	bSeqAbort					:BOOL;		(*Function Abort By Manager*)
	bSeqHomingRequest			:BOOL;		(*FUNCTION Homing Requested BY Manager OR Internal Functions*)
	bSeqWaitOnRequest			:BOOL;		(*Function In Valide State Avaiting For Request Command*)
	bSeqRequest					:BOOL;		(*Request Commnad To Start Function Cycle*)

	bSeqIsHoming					: BOOL;
	bSeqInProgress				:BOOL;		(*Function In Progress With Cycle*)
	bSeqComplete				:BOOL;		(*Function Complete Cycle - Flag Set After Every Cycle Finsh*)
	bSeqDone					:BOOL;		(*Function Sequence Finished With Success - Flag Set For One PLC Cycle*)
	bSeqError						: BOOL;
	nSeqErrorID					: UDINT;

	bAutoHomingAllowed			: BOOL;
	bStationHomed					:BOOL;		(*FUNCTION Homed*)
	bStationNotMoving				:BOOL;		(*Function Parts Are Not Moving*)
	bStationInPause				: BOOL;

	bMachineInError				: BOOL;
	bPassthroughMode				:BOOL;

	stBundleTracking				: ST_BundleTrackingRegister_C715;
	bTrackigDataSync				: BOOL;
	bDisableBottomLimit			: BOOL;

	bSynchroMoveActive			: BOOL;

END_STRUCT
END_TYPE

// ---- DUTs/METS/_StationOperational/C715 Tempalate Example/ST_BundleTrackingRegister_C715.TcDUT
TYPE ST_BundleTrackingRegister_C715 :
STRUCT
	bOuterPresent				: BOOL;
	sOuterTimeStamp			: STRING(30);
	bOuterAligned				: BOOL;
	bLabelApplied				: BOOL;		(* TRUE = label has been printed and applied to Outer *)
	bLabelFormed				: BOOL;
	sLabelBarcode				: T_OUTER_Barcode;
	sConfirmationCode 			: T_MaxString;
	bOCVCreated				: BOOL;
	bOACCreated				: BOOL;
	bOuterIsValid				: BOOL;
	bDumpDataReq			: BOOL;
END_STRUCT
END_TYPE

// ---- DUTs/METS/_StationOperational/E_00_StationStateTemplate.TcDUT
TYPE E_00_StationStateTemplate :
(
	SEQ_00_INIT									:=0,
	SEQ_00_ENABLEDEVICES							:=1,
	SEQ_00_HOMING								:=10,
	SEQ_00_MOVETOHOMEPOS_TRY					:=20,
	SEQ_00_MOVETOHOMEPOS_DONE					:=30,
	SEQ_00_HOMED								:=90,
	SEQ_00_READY									:=100,

	SEQ_00_REQACCEPTED							:=110,

(***************************************************************************)
(**)
(***************************************************************************)

	SEQ_00_COMPLETE_TRY							:=340,
	SEQ_00_COMPLETE								:=350


);
END_TYPE

// ---- DUTs/METS/_StationOperational/Manual Machine/E_OuterPrintStationState.TcDUT
TYPE E_OuterPrintStationState :
(
	STATION_SEQ_INIT:=100,
	STATION_SEQ_TRY_HOMING:=110,
	STATION_SEQ_HOMED:=120,
	STATION_SEQ_READY:=130,

	STATION_SEQ_GATE_DOWN_TRY:=140,
	STATION_SEQ_GATE_DOWN_DONE:=150,

	STATION_SEQ_APPLY_LABEL_TRY:=160,
	STATION_SEQ_APPLY_LABEL_DONE:=170,

	STATION_SEQ_GATE_UP_TRY:=180,
	STATION_SEQ_GATE_UP_DONE:=190,

	STATION_SEQ_COMPLETE_TRY:=200,
	STATION_SEQ_COMPLETE:=210


);
END_TYPE

// ---- DUTs/METS/_StationOperational/Manual Machine/ST_OuterPrintStationStruct.TcDUT
TYPE ST_OuterPrintStationStruct :
STRUCT

	eOuterPrintStationState				: 	E_OuterPrintStationState;

	bStationRequest			: 	BOOL;		(*Request Commnad To Start Function Cycle*)
	bStationWaitOnRequest	:	BOOL;		(*Function In Valide State Avaiting For Request Command*)
	bStationInProgress		: 	BOOL;		(*Function In Progress With Cycle*)
	bStationComplete			: 	BOOL;		(*Function Complete Cycle - Flag Set After Every Cycle Finsh*)

	bStationHomingRequest		:	BOOL;		(*FUNCTION Homing Requested BY Manager OR Internal Functions*)
	bStationHomed					: 	BOOL;		(*FUNCTION Homed*)
	bStationDone					:	BOOL;		(*Function Sequence Finished With Success - Flag Set For One PLC Cycle*)
	bStationAbort					: 	BOOL;		(*Function Abort By Manager*)
	bStationInhibit					: BOOL;

	bStationNotMoving			: 	BOOL;		(*Function Parts Are Not Moving*)

	bPassthroughMode						: BOOL;


	eGateCommand		: E_CYLINDER_Position := E_CYLINDER_Position.STOP;

	bGateInPosition					: BOOL;
	bGateRetractedPosition				: BOOL;
	bGateExtendedPosition				: BOOL;
	bGateIsRetracting					: BOOL;
	bGateIsExtending					: BOOL;
	bGatePositionError					: BOOL;

	bOuterAtApplyPosition					: BOOL;
	bApplyLabel							: BOOL;
	bApplyDone							: BOOL;

	bSkipGate							: BOOL;
END_STRUCT
END_TYPE

// ---- DUTs/METS/_StationOperational/SeqCtrl/ST_STATION_Requests.TcDUT
TYPE ST_STATION_Requests :
STRUCT

	bSeqAbort						:BOOL;		(*Function Abort By Manager*)
	bSeqInhibit						: BOOL;		(*in girafe is like bMachineInError*)
	bSeqHomingRequest			:BOOL;		(*FUNCTION Homing Requested BY Manager OR Internal Functions*)
	bSeqWaitOnRequest			:BOOL;		(*Function In Valide State Avaiting For Request Command*)
	bSeqRequest					:BOOL;		(*Request Commnad To Start Function Cycle*)

END_STRUCT
END_TYPE

// ---- DUTs/METS/_StationOperational/SeqCtrl/ST_STATION_Status.TcDUT
TYPE ST_STATION_Status :
STRUCT

	bSeqIsHoming					: BOOL;
	bStationHomed					:BOOL;		(*FUNCTION Homed*)
	bSeqInProgress				:BOOL;		(*Function In Progress With Cycle*)
	bSeqComplete				:BOOL;		(*Function Complete Cycle - Flag Set After Every Cycle Finsh*)
	bSeqDone					:BOOL;		(*Function Sequence Finished With Success - Flag Set For One PLC Cycle*)
	bStationNotMoving				:BOOL;		(*Function Parts Are Not Moving*)

	bSeqError						: BOOL;
	nSeqErrorID					: UDINT;

END_STRUCT
END_TYPE

// ---- DUTs/METS/_StationOperational/ST_00_StationStructTemplate.TcDUT
TYPE ST_00_StationStructTemplate :
STRUCT

	e00SeqState		: E_00_StationStateTemplate;

	REQ				: ST_STATION_Requests;
	STAT				: ST_STATION_Status;

(*Variable examles only*)
(*
	bPassthroughMode			:BOOL;

	stBundleTracking				: ST_BundleTrackingRegister;
	bTrigCamera					: BOOL;
	bCameraDone					: BOOL;


*)

END_STRUCT
END_TYPE

// ---- DUTs/Test_DUTs/ST_DuplicateInfo.TcDUT
TYPE ST_DuplicateInfo :
STRUCT
	value 			: T_MaxString;
	nOuterIndex 	: UINT;
	PackIndex 		: UINT;
END_STRUCT
END_TYPE

// ---- DUTs/Test_DUTs/ST_FBinside.TcDUT
TYPE ST_FBinside :
STRUCT
	aTONs		: ARRAY[1..10] OF TON;
	aTOFs		: ARRAY[1..10] OF TOF;
END_STRUCT
END_TYPE

// ---- DUTs/Test_DUTs/ST_LAB_CaseData.TcDUT
TYPE ST_LAB_CaseData :
STRUCT
	aOuters		: ARRAY[1..50] OF ST_LAB_OuterData;
END_STRUCT
END_TYPE

// ---- DUTs/Test_DUTs/ST_LAB_OuterData.TcDUT
TYPE ST_LAB_OuterData :
STRUCT
	sOuterCode			: T_MaxString;
	nOutersStatus		: INT;
	nOuterRejectID		: UINT;
	
	aPacks				: ARRAY[1..10] OF ST_LAB_PackData;
END_STRUCT
END_TYPE

// ---- DUTs/Test_DUTs/ST_LAB_PackData.TcDUT
TYPE ST_LAB_PackData :
STRUCT
	sPackCode			: T_MaxString;
	nPackStatus			: INT;
	nPackRejectID		: UINT;
END_STRUCT
END_TYPE

// ---- GVLs/CodeAI.TcGVL
{attribute 'Tc2GvlVarNames'}
VAR_GLOBAL
	eCodeAIType							: E_CodeAIType;
	


END_VAR

// ---- GVLs/gConstants.TcGVL
{attribute 'Tc2GvlVarNames'}
//{warning 'CONVERSION MESSAGE: This text contained unprintable characters, that have been deleted'.}
VAR_GLOBAL CONSTANT

	(* sub-folders for  directory *)
	cSYSTEM_FOLDER_LIMIT				: INT :=20;

	(*cBASE_FOLDER_ARR					: ARRAY[1..cSYSTEM_FOLDER_LIMIT] OF T_FolderName :=[
			(*01*)'Bridge\',	(*02*)'Bridge\Archive\',	(*03*)'Bridge\Restore\',
			(*04*)'CAC\',		(*05*)'CAC\Archive\',		(*06*)'CAC\Error\',	(*07*)'CAC\Restore\', 	(*08*)'CAC\Restore\Archive\',
			(*09*)'CHM\',		(*10*)'CHM\Archive\',		(*11*)'CHM\Error\',	(*12*)'CHM\OK\',		(*13*)'CHM\Commissioning_Mode\',
			(*14*)'HMI\',
			(*15*)'KPI\',		(*16*)'KPI\Archive\',		(*17*)'KPI\Shift\',	(*18*)'KPI\ProdOrder\',
			(*19*)'OAC\',		(*20*)'OAC\Error\',
			(*21*)'OCV\',		(*22*)'OCV\Error\',
			(*23*)'OHM\',		(*24*)'OHM\Archive\',		(*25*)'OHM\Error\',	(*26*)'OHM\OK\',		(*27*)'OHM\Pending\',
			(*28*)'PCM\',		(*29*)'PCM\Archive\',		(*30*)'PCM\Error\',	(*31*)'PCM\Incoming\',
			(*32*)'PAC\',
			(*33*)'PHM\',		(*34*)'PHM\Archive\',		(*35*)'PHM\Error\',	(*36*)'PHM\OK\',
			(*37*)'Settings\',	(*38*)'Settings\Backups\',
			(*39*)'Templates\',
			(*40*)'Orca\',
			(*41*)'SystemLog\',
			(*42*)'Cameras\',
			(*43*)'ArchiveDB\'];*)
			
cMETS_CORE_FOLDERS					: ARRAY[1..cSYSTEM_FOLDER_LIMIT] OF T_FolderName :=[
			(*01*)'CHM\',		(*02*)'CHM\Archive\',		(*03*)'CHM\Error\',		(*04*)'CHM\OK\',		(*05*)'CHM\Commissioning_Mode\',	(*06*)'CHM\Restore\',
			(*07*)'PCM\',		(*08*)'PCM\Archive\',		(*09*)'PCM\Error\',		(*10*)'PCM\Incoming\',
			(*11*)'Settings\',	(*12*)'Settings\Backups\',	(*13*)'Settings\Recipe\',
			(*14*)'Cameras\',
			(*15*)'Printers\',	(*16*)'Printers\Templates'];
			
cMETS_AUX_FOLDERS					: ARRAY[1..cSYSTEM_FOLDER_LIMIT] OF T_FolderName :=[
			(*01*)'CAC\',		(*02*)'CAC\Archive\',		(*03*)'CAC\Error\',		(*04*)'CAC\Restored\',
			(*05*)'OAC\',		(*06*)'OAC\Error\',			(*07*)'OAC\Empty\',
			(*08*)'OCV\',		(*09*)'OCV\Error\',			(*10*)'OCV\Empty\',
			(*11*)'SystemLog\',
			(*12*)'ArchiveDB\',
			(*13*)'BridgeApp\Bridge_Core\',
			(*14*)'LoggerApp\Service\',
			(*15*)'WebHMI\',
			(*16*)'DeleteArchiveTool\'];
			
			
	cME_ARCHIVE_ACTION 					: ARRAY[1..3] OF STRING :=[
			(*01*)'Archive', 	(*02*)'DeleteTime', 		(*03*)'DeleteItem'] ;

	cMAX_HMI_DISPLAYS					: INT:=2;
	cMAX_HMI_SERIALCODE_LENGHT			: INT := 33;

	cDISABLE_LOG						: BOOL := FALSE;
	cDISABLE_ALARMS						: BOOL := FALSE;
	cMAX_ALARM_GROUP					: T_PositiveINT:=7;
	cMAX_MESSAGE_NUMBER					: T_PositiveINT:=255;
	cMAX_DISPLAY_ALARMS					: T_PositiveINT := 100;

	cMAX_PACK_INFEED_QUEUE				: T_PositiveINT := 80;  (*IMPORTANT index needs to by grater than max value form aPackCodeMapping20*)
	cMAX_HMI_PACK_INFEED_QUEUE			: T_PositiveINT :=100;	(*must be FIXED 100 for HMI and bigger then cMAX_PACK_INFEED_QUEUE*)

	cMAX_INTERMEDIATE_CODE_QUEUE		: T_PositiveINT := 10;
	(*cMAX_TRACE_UNIT_QUEUE				: UINT := 5;
	cMAX_PACK_REJECTED_QUEUE			: UINT := 30;*)

	cMAX_PACKCODE_LENGHT				: T_PositiveINT := 60;
	cMAX_HMI_PACKCODE_LENGHT			: T_PositiveINT := 67;

	cMAX_PACKS_PER_OUTER				: T_PositiveINT :=10;
	cMAX_HMI_PACKS_PER_OUTER			: T_PositiveINT :=20;	(*must be FIXED 20 for HMI and bigger then cMAX_PACKS_PER_OUTER*)

	cMAX_OUTER_STATUS_QUEUE				: T_PositiveINT := 50;
	cMAX_INFEED_QUEUE					: T_PositiveINT :=100;

	cMAX_OUTERS_PER_CASE 				: T_PositiveINT := 70;
	cMAX_HMI_OUTERS_PER_CASE 			: T_PositiveINT := 100;	(*must be FIXED  100 for HM and bigger then cMAX_OUTERS_PER_CASE*)

	cMAX_PACK_PER_CASE 					: T_PositiveINT := 840;	(*must be cMAX_PACKS_PER_OUTER* cMAX_OUTERS_PER_CASE*)

	cMAX_SIDEFLEX_QUEUE					: T_PositiveINT :=10;
	cMAX_CASE_QUEUE						: T_PositiveINT :=4;
	cMAX_FAILED_CASE_QUEUE				: T_PositiveINT :=10;
	cMAX_VERIFIED_CASE_QUEUE			: T_PositiveINT :=10;
	cMAX_LAST_CASE_BARCODES				: T_PositiveINT := 10;

	cMAX_CHM_PACKID_LENGHT				: T_PositiveINT := 60;
	cMAX_CHM_OUTERID_LENGHT				: T_PositiveINT := 60;
	cMAX_CHM_CASEID_LENGHT				: T_PositiveINT := 25;

	cSHIFTNUMBER						: T_PositiveINT := 4;

	cCODE_OVERWIRTTEN					: STRING(12) := '************';
	cCASE_PACKER_REJECT					: STRING := 'CASE_REJECT_BY_CASEPACKER';
	cMAX_REJECT_REASON					: T_PositiveINT := 80;
	cXML_HEADER							: STRING :=   '<?xml version="1.0" encoding="utf-8"?>$R$N';

	cPARAMETER_STORAGE_SIZE				: T_PositiveINT := 25;	(*  *)


	cMAX_ETHERCAT_SLAVES				: T_PositiveINT := 63; 	(* tabel start with 0 and 64 elemnts *)
	cMAX_PNOZ_ELEMENTS					: T_PositiveINT := 20;
	cMAX_PROFINET_MASTERS	      		: T_PositiveINT := 2; 		(* Must always be set min to 2*)
	cMAX_PROFINET_DRIVES        		: T_PositiveINT := 8;		(* Must always be set min to 8*)
	cMAX_ANALOG_DRIVERS					: T_PositiveINT := 2; 		(* Must always be set min to 2*)
	cMAX_MC2_DRIVES						: T_PositiveINT := 2;
	cMAX_CYLINDERS						: T_PositiveINT := 12;		(*Must always be set min to 3*)
	cMAX_PRINTER_NUMBER           		: T_PositiveINT := 6;		(*Must always be set min to 6*)
	cMAX_HAND_SCANNERS					: T_PositiveINT := 2; 		(*Must always be set min to 2*)
	cMAX_CAMS							: T_PositiveINT := 1;
	cMAX_ENCODER						: T_PositiveINT := 1;
	cMAX_CAMERA_PROG_NUMBER				: T_PositiveINT := 5;
	cMAX_CAMERA_NUMBER					: T_PositiveINT :=12;		(*Must always be set min to 12*)
	cOUT_CAMERA_GROUP					: T_PositiveINT:=9;
	cCS_CAMERA_GROUP					: T_PositiveINT:=12;
	cPLAS_CAMERA_OFF_DELAY				: TIME:= T#10S;

	cDOT_CHAR 							: T_Char := '.';
	cTAB_CHAR 							: T_Char := '$09';
	cLF_CHAR 							: T_Char := '$0A';
	cCR_CHAR							: T_Char := '$0D';

	cHALF_SECOND						: TIME := t#0.5s;
	cONE_SECOND							: TIME := T#1s;
	cTWO_SECONDS						: TIME := T#2s;
	cTHREE_SECONDS						: TIME := T#3s;
	cFIVE_SECONDS						: TIME := t#5s;
	cTEN_SECONDS						: TIME := t#10s;

	cONE_MINUTE							: TIME := t#1m;
	cFIVE_MINUTES						: TIME := T#5m;
	cONE_HOUR							: TIME := T#1h;

	(* File handling *)
	cFAILED_INVALID_INDEX_GROUP			: DWORD :=  16#702;
	cFAILED_INVALID_INDEX_OFFSET		: DWORD :=  16#703;
	cFAILED_OBJECT_NOT_FOUND			: DWORD :=  16#70C;
	cFAILED_OBJECT_ALREADY_EXIST		: DWORD :=  16#70F;
	cFAILED_NO_MORE_FILE_HANDLES		: DWORD :=  16#716;
	cFAILED_ACCESS_DENIED				: DWORD :=  16#723;
	
	(* File handling *)
	//cFAILED_INVALID_DATA				: DWORD :=  16#703;
	//cFAILED_FILE_NOT_FOUND			: DWORD :=  16#70C;
	//cFAILED_NO_MORE_FILE_HANDLES		: DWORD :=  16#716;
	cMAX_FILE_BUFFER					: T_PositiveINT := 32767;(*10000;*)

	cNUMBER_DEFINED_AI_TYPES			: T_PositiveINT :=14;
	cMAX_VALIDATION_ITEMS				: T_PositiveINT :=10;

	(*cUSE_INTERMEDIATE_BARCODE_VALIDATION	: BOOL := TRUE;*)

	cMAX_CAMERA_TYPES					: T_PositiveINT :=15;

	cACQUISITION_TIMER					: ARRAY[0..cMAX_CAMERA_TYPES] OF TIME :=[
			(*Number of array elemnts must match to number of elemnts in E_SCANNER_DeviceType*)
			(*E_MV_None*)T#0ms,
			(*E_MV_420_FULL*)T#26ms,			(*E_MV_420_HALF*)T#12ms,
			(*E_MV_440SR_FULL*)T#18ms, 		(*E_MV_440SR_HALF*)T#12ms,
			(*E_MV_440HR_FULL*)T#52ms, 		(*E_MV_440HR_HALF*)T#30ms,
			(*E_MV_440UR_FULL*)T#50ms, 		(*E_MV_440UR_HALF*)T#33ms,
			(*E_MV_540S_FULL*)T#24ms, 			(*E_MV_540S_HALF*)T#12ms,
			(*E_MV_540H_FULL*)T#24ms, 			(*E_MV_540H_HALF*)T#12ms,
			(*E_MV_560U_FULL*)T#24ms, 			(*E_MV_560U_HALF*)T#12ms,
			(*E_V_430F_FULL*)T#18ms];


END_VAR

// ---- GVLs/GVL.TcGVL
{attribute 'qualified_only'}
VAR_GLOBAL
	bTriggerButton		AT %I* : BOOL;			
	bTriggerOutput		AT %Q* : BOOL;		


	// Hikrobot Control Commands

	aHikrobotCtrlCommands				: ARRAY[1..20] OF STRING(40) :=[
		(*start user params 0*) 		'<Set,UserStart,0>',
		(*start user params 1*) 		'<Set,UserStart,1>',
		(*start user params 2*) 		'<Set,UserStart,2>',
		(*execute self adjustement*) 	'<Exec,Tune>',
		(*start reading codes*) 		'<Set,Acq,1><Set,UserStart,3>',
		(*stop reading codes*) 			'<Set,Acq,0>',
		(*camera reboot*) 				'<Exec,Reboot>',
		(*camera reboot*) 				'<Get,RunMode>',
		(*camera reboot*) 				'<Set,RunMode,2>',
		(*camera reboot*) 				'<Set,RunMode,0>'
];


	aTCPxStrings						: ARRAY[0..20] OF T_MaxString;
	aTCPxStringsReply					: ARRAY[0..20] OF T_MaxString;

END_VAR

// ---- GVLs/GVL_HIKROBOT_COMMANDS.TcGVL
{attribute 'qualified_only'}
VAR_GLOBAL
END_VAR

// ---- GVLs/GVL_test.TcGVL
{attribute 'qualified_only'}
VAR_GLOBAL
	
	//aCase	: ARRAY[1..3] OF ST_LAB_OuterData ;
	stCase		:	ST_LAB_CaseData; 
	stCaseFull	:	ST_LAB_CaseData; 

	
	nMax_Outers			: UINT := 50;
	nMax_Packs			: UINT := 10;


	
// 	aInputArray		: ARRAY[1..3, 1..3] OF T_MaxString := [ 
// 	['PACK01OUTER1', 'PACK02OUTER1', 'PACK03OUTER1'],
// 	['PACK01OUTER2', 'PACK02OUTER2', 'PACK03OUTER2'],
// 	['PACK01OUTER3', 'PACK02OUTER3', 'PACK03OUTER3']
// 	];


	stFBinside		: ST_FBinside;

END_VAR

// ---- POUs/PRG_TEST.TcPOU
PROGRAM PRG_TEST
VAR
	//fbCaseDuplicatCheckTests			: FB_CASE_DuplicatCheckTests;
	//fbCaseDuplicateUpdateToDBTests	: FB_CASE_DuplicateUpdateToDBTests;
	//fbCaseFinaliseDataTests				: FB_CASE_FinaliseDataTests;
	//fbCaseInitialiseData_Test 			: FB_CASE_InitialiseDataTests;
	fbCaseValidateContentTests		: FB_CASE_ValidateContentTests;
	
END_VAR

//===================================================
//UNIT TEST EXECUTION

TcUnit.RUN();

//===================================================
//MANUAL TEST EXECUTION

PRG_CASE_DuplicatCheckManual();
PRG_CASE_DuplicateUpdateToDBManual();
PRG_CASE_FinaliseDataManual();
PRG_CASE_InitialiseDataManual();
PRG_CASE_ValidateContentManual();



//===================================================
//TESTS for FB references
//PRG_Reference_POU();

END_PROGRAM

// ---- POUs/TcUnit/FB_CASE_ValidateContentTests/FB_CASE_ValidateContentTests.TcPOU
FUNCTION_BLOCK FB_CASE_ValidateContentTests EXTENDS TcUnit.FB_TestSuite

VAR
	
(* General data *)
	stCTDateTime_tests					: ST_SYSTEM_DateTime;	
	stProductInstruction_tests			: ST_PCM_Status;
	nSecquentionalCounter_tests			: UDINT;
	stCodeInfo_Outer_tests				: ST_CodeInfo;
	stCaseRejectReasons_tests			: ST_RejectReasonsForCase;
	stRejectReasonsForOuter_tests		: ST_RejectReasonsForOuter;
	stOuterDataNotFound_tests			: ST_RejectItems;

(* 01.Main tests container *)

	stProductInstruction_test_0101		: ST_PCM_Status;
	stCACData_test_0101 				: ST_CAC_Data;
		
	stCACData_tests 					: ST_CAC_Data;
(* 02.DataConsistancy tests container *)
	stProductInstruction_test_0201		: ST_PCM_Status;
	stCACData_test_0201 				: ST_CAC_Data;
	sRejectCode_test_0201				: T_MaxString;
	
	stProductInstruction_test_0202		: ST_PCM_Status;
	stCACData_test_0202 				: ST_CAC_Data;
	sRejectCode_test_0202				: T_MaxString;	
	
	
	stProductInstruction_test_0203		: ST_PCM_Status;
	stCACData_test_0203 				: ST_CAC_Data;
	sRejectCode_test_0203				: T_MaxString;
	
	stProductInstruction_test_0204		: ST_PCM_Status;
	stCACData_test_0204 				: ST_CAC_Data;
	sRejectCode_test_0204				: T_MaxString;

	
	stProductInstruction_test_0205		: ST_PCM_Status;
	stCACData_test_0205 				: ST_CAC_Data;
	sRejectCode_test_0205				: T_MaxString;
	
	stProductInstruction_test_0206		: ST_PCM_Status;
	stCACData_test_0206 				: ST_CAC_Data;
	sRejectCode_test_0206				: T_MaxString;

(* 03.NumberOfOuters tests container *)
	stProductInstruction_test_0301		: ST_PCM_Status;
	stCACData_test_0301 				: ST_CAC_Data;
	sRejectCode_test_0301				: T_MaxString;
	
	stProductInstruction_test_0302		: ST_PCM_Status;
	stCACData_test_0302 				: ST_CAC_Data;
	sRejectCode_test_0302				: T_MaxString;
	
	stProductInstruction_test_0303		: ST_PCM_Status;
	stCACData_test_0303 				: ST_CAC_Data;
	sRejectCode_test_0303				: T_MaxString;
	
(* 04.OuterAggrDissable tests container *)
	stProductInstruction_test_0401		: ST_PCM_Status;
	stCACData_test_0401 				: ST_CAC_Data;
	sRejectCode_test_0401				: T_MaxString;
	
	stProductInstruction_test_0402		: ST_PCM_Status;
	stCACData_test_0402 				: ST_CAC_Data;
	sRejectCode_test_0402				: T_MaxString;

(* 05.OuterAggrEnable tests container *)
	stProductInstruction_test_0501		: ST_PCM_Status;
	stCACData_test_0501 				: ST_CAC_Data;
	sRejectCode_test_0501				: T_MaxString;
	
	stProductInstruction_test_0502		: ST_PCM_Status;
	stCACData_test_0502 				: ST_CAC_Data;
	sRejectCode_test_0502				: T_MaxString;

(* 06.DuplicateHandler tests container *)
	
	stProductInstruction_test_0601		: ST_PCM_Status;
	stCACData_test_0601 				: ST_CAC_Data;
	sRejectCode_test_0601				: T_MaxString;
	
	stCACData_test_0602 				: ST_CAC_Data;
	stProductInstruction_test_0602		: ST_PCM_Status;
	sRejectCode_test_0602				: T_MaxString;
	
(* 07.OACmissing tests container *)
	
	stProductInstruction_test_0701		: ST_PCM_Status;
	stCACData_test_0701 				: ST_CAC_Data;
	sRejectCode_test_0701				: T_MaxString;
	
	stCACData_test_0702 				: ST_CAC_Data;
	stProductInstruction_test_0702		: ST_PCM_Status;
	sRejectCode_test_0702				: T_MaxString;
	
	sRejectCode_tets					: T_MaxString;
	
END_VAR


//==============================================================
//01.Main
//==============================================================
main01_bExecuteFalseNoAction();
//==============================================================
//02.DataConsistancy
//==============================================================
dataConsistancy01_NumOfOutersWrong();
dataConsistancy02_NumOfOutersExceedcMAX_Outers();
dataConsistancy03_ValidationCodeNotFoundInInfeedQueue();
dataConsistancy04_OuterCodeVal_IndexErrorFound();
dataConsistancy05_NumberOfOutersToSmall();
dataConsistancy06_NumberOfOutersToBig();

//==============================================================
//03.NumberOfOuters
//==============================================================
numberOfOuters01_ValueToLittlebErrorTrue();
numberOfOuters02_ValueGraterErrorTrue();
numberOfOuters03_ValueToLittlebErrorTrueRejectCodeWright();

//==============================================================
//04.OuterAggrDissable
//==============================================================
outerAggrDissable01_sRejectCodeOK();

//==============================================================
//05.OuterAggrEnable
//==============================================================
outerAggrEnable01_PacksPerOuterZero();
outerAggrEnable02_PacksPerCaseZero();


//==============================================================
//06.DuplicatesHandler
//==============================================================
duplicateHandler01_OuterDuplicatebErrorTrue();
duplicateHandler02_PackDuplicatebErrorTrue();

//==============================================================
//07.OACmissing
//==============================================================
oacMissing01nErrorID21();

METHOD INTERNAL dataConsistancy01_NumOfOutersWrong
VAR
	//fbCaseTest			: FB_CASE_ValidateContent;
	bDone				: BOOL;
	bBusy				: BOOL;
	bError				: BOOL;
	nErrorID 			: UDINT;
	nValidationIndex	: INT;
	
	eLastState			: E_CAC_State;
			
END_VAR

VAR_INST
	fbCaseTest0201				: FB_CASE_ValidateContent;
	rTrig0201					: R_TRIG;
	nCycles0201					: INT;
	
END_VAR

//Data initialization
TestInit(stCACData:= stCACData_test_0201, stProductInstruction:= stProductInstruction_test_0201);

//Change some data for test scenario below
stCACData_test_0201.NumberOfOuters := stCACData_test_0201.NumberOfOuters - 2;
	
TcUnit.TEST('dataConsistancy01_NumOfOutersWrong');


fbCaseTest0201(
	bExecute:= TRUE, 
	bIsDuplicateOuters:= FALSE, 
	bIsDuplicatePacks:= FALSE, 
	stCTDateTime:= stCTDateTime_tests, 
	stOuterDataNotFound:= stRejectReasonsForOuter_tests.stOuterDataNotFound, 
	stProductInstruction:= stProductInstruction_test_0201, 
	nSecquentionalCounter:= nSecquentionalCounter_tests, 
	stCodeInfo_Outer:= stCodeInfo_Outer_tests, 
	stCaseRejectReasons:= stCaseRejectReasons_tests, 
	stCACData:= stCACData_test_0201, 
	bDone=> bDone, 
	bBusy=> bBusy, 
	bError=> bError, 
	nErrorID=> nErrorID, 
	sRejectCode=> sRejectCode_test_0201, 
	nValidationIndex=> nValidationIndex
);
	
rTrig0201(CLK:= fbCaseTest0201.bDone);
nCycles0201 := nCycles0201 + 1;	

IF rTrig0201.Q THEN	
		
	AssertEquals_BOOL(Expected 	:= TRUE,
					  Actual 	:= bError,
					  Message 	:= 'Wrong number of outers not detected'
	);
	
	AssertEquals_STRING(Expected := 'XXVAL048XX',
						Actual := TO_STRING(fbCaseTest0201.sRejectCode),
						Message := 'Wrong value of nErrorID'
	);
	
	TEST_FINISHED();
	
ELSIF nCycles0201 > 50 THEN
	
	AssertTrue(Condition := TRUE,
			   Message 	 := 'Timeout dataConsistancy01_NumOfOutersWrong'
	);	 
	TEST_FINISHED();
END_IF
END_METHOD

METHOD INTERNAL dataConsistancy02_NumOfOutersExceedcMAX_Outers
VAR
	//fbCaseTest			: FB_CASE_ValidateContent;
	bDone				: BOOL;
	bBusy				: BOOL;
	bError				: BOOL;
	nErrorID 			: UDINT;
	nValidationIndex	: INT;
	
	eLastState			: E_CAC_State;
			
END_VAR

VAR_INST
	fbCaseTest0202				: FB_CASE_ValidateContent;
	rTrig0202					: R_TRIG;
	nCycles0202					: INT;
	
END_VAR

//Data initialization
TestInit(stCACData:= stCACData_test_0202, stProductInstruction:= stProductInstruction_test_0202);

//Change some data for test scenario below
stCACData_test_0202.NumberOfOuters := - 1;
	
TcUnit.TEST('dataConsistancy02_NumOfOutersExceedcMAX_Outers');


fbCaseTest0202(
	bExecute:= TRUE, 
	bIsDuplicateOuters:= FALSE, 
	bIsDuplicatePacks:= FALSE, 
	stCTDateTime:= stCTDateTime_tests, 
	stOuterDataNotFound:= stRejectReasonsForOuter_tests.stOuterDataNotFound, 
	stProductInstruction:= stProductInstruction_test_0202, 
	nSecquentionalCounter:= nSecquentionalCounter_tests, 
	stCodeInfo_Outer:= stCodeInfo_Outer_tests, 
	stCaseRejectReasons:= stCaseRejectReasons_tests, 
	stCACData:= stCACData_test_0202, 
	bDone=> bDone, 
	bBusy=> bBusy, 
	bError=> bError, 
	nErrorID=> nErrorID, 
	sRejectCode=> sRejectCode_test_0202, 
	nValidationIndex=> nValidationIndex
);
	
rTrig0202(CLK:= fbCaseTest0202.bDone);
nCycles0202 := nCycles0202 + 1;	

IF rTrig0202.Q THEN	
		
	AssertEquals_UDINT(Expected := 11,
                   	   Actual 	:= fbCaseTest0202.nErrorID,
                   	   Message 	:= 'nErrorID value wrong');
	
	TEST_FINISHED();
	
ELSIF nCycles0202 > 50 THEN
	
	AssertTrue(Condition := TRUE,
			   Message 	 := 'Timeout dataConsistancy02_NumOfOutersExceedcMAX_Outers'
	);	 
	TEST_FINISHED();
END_IF
END_METHOD

METHOD INTERNAL dataConsistancy03_ValidationCodeNotFoundInInfeedQueue
VAR
	//fbCaseTest			: FB_CASE_ValidateContent;
	bDone				: BOOL;
	bBusy				: BOOL;
	bError				: BOOL;
	nErrorID 			: UDINT;
	nValidationIndex	: INT;
	
	eLastState			: E_CAC_State;
			
END_VAR

VAR_INST
	fbCaseTest0203				: FB_CASE_ValidateContent;
	rTrig0203					: R_TRIG;
	nCycles0203					: INT;
	
END_VAR

//Data initialization
TestInit(stCACData:= stCACData_test_0203, stProductInstruction:= stProductInstruction_test_0203);

//Change some data for test scenario below
stCACData_test_0203.NumberOfOuters := - 2;
	
TcUnit.TEST('dataConsistancy03_ValidationCodeNotFoundInInfeedQueue');


fbCaseTest0203(
	bExecute:= TRUE, 
	bIsDuplicateOuters:= FALSE, 
	bIsDuplicatePacks:= FALSE, 
	stCTDateTime:= stCTDateTime_tests, 
	stOuterDataNotFound:= stRejectReasonsForOuter_tests.stOuterDataNotFound, 
	stProductInstruction:= stProductInstruction_test_0203, 
	nSecquentionalCounter:= nSecquentionalCounter_tests, 
	stCodeInfo_Outer:= stCodeInfo_Outer_tests, 
	stCaseRejectReasons:= stCaseRejectReasons_tests, 
	stCACData:= stCACData_test_0203, 
	bDone=> bDone, 
	bBusy=> bBusy, 
	bError=> bError, 
	nErrorID=> nErrorID, 
	sRejectCode=> sRejectCode_test_0203, 
	nValidationIndex=> nValidationIndex
);
	
rTrig0203(CLK:= fbCaseTest0203.bDone);
nCycles0203 := nCycles0203 + 1;	

IF rTrig0203.Q THEN	
		
	AssertEquals_UDINT(Expected := 12,
                   	   Actual 	:= fbCaseTest0203.nErrorID,
                   	   Message 	:= 'nErrorID value wrong');
	
	TEST_FINISHED();
	
ELSIF nCycles0203 > 50 THEN
	
	AssertTrue(Condition := TRUE,
			   Message 	 := 'Timeout dataConsistancy03_ValidationCodeNotFoundInInfeedQueue'
	);	 
	TEST_FINISHED();
END_IF
END_METHOD

METHOD INTERNAL dataConsistancy04_OuterCodeVal_IndexErrorFound
VAR
	//fbCaseTest			: FB_CASE_ValidateContent;
	bDone				: BOOL;
	bBusy				: BOOL;
	bError				: BOOL;
	nErrorID 			: UDINT;
	nValidationIndex	: INT;
	
	eLastState			: E_CAC_State;
			
END_VAR

VAR_INST
	fbCaseTest0204				: FB_CASE_ValidateContent;
	rTrig0204					: R_TRIG;
	nCycles0204					: INT;
	
END_VAR

//Data initialization
TestInit(stCACData:= stCACData_test_0204, stProductInstruction:= stProductInstruction_test_0204);

//Change some data for test scenario below
stCACData_test_0204.NumberOfOuters := - 3;
	
TcUnit.TEST('dataConsistancy04_OuterCodeVal_IndexErrorFound');


fbCaseTest0204(
	bExecute:= TRUE, 
	bIsDuplicateOuters:= FALSE, 
	bIsDuplicatePacks:= FALSE, 
	stCTDateTime:= stCTDateTime_tests, 
	stOuterDataNotFound:= stRejectReasonsForOuter_tests.stOuterDataNotFound, 
	stProductInstruction:= stProductInstruction_test_0204, 
	nSecquentionalCounter:= nSecquentionalCounter_tests, 
	stCodeInfo_Outer:= stCodeInfo_Outer_tests, 
	stCaseRejectReasons:= stCaseRejectReasons_tests, 
	stCACData:= stCACData_test_0204, 
	bDone=> bDone, 
	bBusy=> bBusy, 
	bError=> bError, 
	nErrorID=> nErrorID, 
	sRejectCode=> sRejectCode_test_0204, 
	nValidationIndex=> nValidationIndex
);
	
rTrig0204(CLK:= fbCaseTest0204.bDone);
nCycles0204 := nCycles0204 + 1;	

IF rTrig0204.Q THEN	
		
	AssertEquals_UDINT(Expected := 13,
                   	   Actual 	:= fbCaseTest0204.nErrorID,
                   	   Message 	:= 'nErrorID value wrong');
	
	TEST_FINISHED();
	
ELSIF nCycles0204 > 50 THEN
	
	AssertTrue(Condition := TRUE,
			   Message 	 := 'Timeout dataConsistancy04_OuterCodeVal_IndexErrorFound'
	);	 
	TEST_FINISHED();
END_IF
END_METHOD

METHOD INTERNAL dataConsistancy05_NumberOfOutersToSmall
VAR
	//fbCaseTest			: FB_CASE_ValidateContent;
	bDone				: BOOL;
	bBusy				: BOOL;
	bError				: BOOL;
	nErrorID 			: UDINT;
	nValidationIndex	: INT;
	
	eLastState			: E_CAC_State;
			
END_VAR

VAR_INST
	fbCaseTest0205				: FB_CASE_ValidateContent;
	rTrig0205					: R_TRIG;
	nCycles0205					: INT;
	
END_VAR

//Data initialization
TestInit(stCACData:= stCACData_test_0205, stProductInstruction:= stProductInstruction_test_0205);

//Change some data for test scenario below
stCACData_test_0205.NumberOfOuters := 25;
	
TcUnit.TEST('dataConsistancy05_NumberOfOutersToSmall');


fbCaseTest0205(
	bExecute:= TRUE, 
	bIsDuplicateOuters:= FALSE, 
	bIsDuplicatePacks:= FALSE, 
	stCTDateTime:= stCTDateTime_tests, 
	stOuterDataNotFound:= stRejectReasonsForOuter_tests.stOuterDataNotFound, 
	stProductInstruction:= stProductInstruction_test_0205, 
	nSecquentionalCounter:= nSecquentionalCounter_tests, 
	stCodeInfo_Outer:= stCodeInfo_Outer_tests, 
	stCaseRejectReasons:= stCaseRejectReasons_tests, 
	stCACData:= stCACData_test_0205, 
	bDone=> bDone, 
	bBusy=> bBusy, 
	bError=> bError, 
	nErrorID=> nErrorID, 
	sRejectCode=> sRejectCode_test_0205, 
	nValidationIndex=> nValidationIndex
);
	
rTrig0205(CLK:= fbCaseTest0205.bDone);
nCycles0205 := nCycles0205 + 1;	

IF rTrig0205.Q THEN	
		
	AssertEquals_UDINT(Expected := 14,
                   	   Actual 	:= fbCaseTest0205.nErrorID,
                   	   Message 	:= 'nErrorID value wrong');
	
	TEST_FINISHED();
	
ELSIF nCycles0205 > 50 THEN
	
	AssertTrue(Condition := TRUE,
			   Message 	 := 'Timeout dataConsistancy05_NumberOfOutersToSmall'
	);	 
	TEST_FINISHED();
END_IF
END_METHOD

METHOD INTERNAL dataConsistancy06_NumberOfOutersToBig
VAR
	//fbCaseTest			: FB_CASE_ValidateContent;
	bDone				: BOOL;
	bBusy				: BOOL;
	bError				: BOOL;
	nErrorID 			: UDINT;
	nValidationIndex	: INT;
	
	eLastState			: E_CAC_State;
			
END_VAR

VAR_INST
	fbCaseTest0206				: FB_CASE_ValidateContent;
	rTrig0206					: R_TRIG;
	nCycles0206					: INT;
	
END_VAR

//Data initialization
TestInit(stCACData:= stCACData_test_0206, stProductInstruction:= stProductInstruction_test_0206);

//Change some data for test scenario below
stCACData_test_0206.NumberOfOuters := 69;
	
TcUnit.TEST('dataConsistancy06_NumberOfOutersToBig');


fbCaseTest0206(
	bExecute:= TRUE, 
	bIsDuplicateOuters:= FALSE, 
	bIsDuplicatePacks:= FALSE, 
	stCTDateTime:= stCTDateTime_tests, 
	stOuterDataNotFound:= stRejectReasonsForOuter_tests.stOuterDataNotFound, 
	stProductInstruction:= stProductInstruction_test_0206, 
	nSecquentionalCounter:= nSecquentionalCounter_tests, 
	stCodeInfo_Outer:= stCodeInfo_Outer_tests, 
	stCaseRejectReasons:= stCaseRejectReasons_tests, 
	stCACData:= stCACData_test_0206, 
	bDone=> bDone, 
	bBusy=> bBusy, 
	bError=> bError, 
	nErrorID=> nErrorID, 
	sRejectCode=> sRejectCode_test_0206, 
	nValidationIndex=> nValidationIndex
);
	
rTrig0206(CLK:= fbCaseTest0206.bDone);
nCycles0206 := nCycles0206 + 1;	

IF rTrig0206.Q THEN	
		
	AssertEquals_UDINT(Expected := 15,
                   	   Actual 	:= fbCaseTest0206.nErrorID,
                   	   Message 	:= 'nErrorID value wrong');
	
	TEST_FINISHED();
	
ELSIF nCycles0206 > 50 THEN
	
	AssertTrue(Condition := TRUE,
			   Message 	 := 'Timeout dataConsistancy06_NumberOfOutersToBig'
	);	 
	TEST_FINISHED();
END_IF
END_METHOD

METHOD INTERNAL duplicateHandler01_OuterDuplicatebErrorTrue
VAR
	//fbCaseTest			: FB_CASE_ValidateContent;
	bDone				: BOOL;
	bBusy				: BOOL;
	bError				: BOOL;
	nErrorID 			: UDINT;
	nValidationIndex	: INT;
	
	eLastState			: E_CAC_State;
			
END_VAR

VAR_INST
	fbCaseTest0601				: FB_CASE_ValidateContent;
	fTrig						: F_TRIG;	
	rTrig						: R_TRIG;
	nCycles						: INT;
	
END_VAR

//Data initialization
TestInit(stCACData:= stCACData_test_0601, stProductInstruction:= stProductInstruction_test_0601);

//Change some data for test scenario below
//stCACData_test_0303.NumberOfOuters := 51;

	
TcUnit.TEST('duplicateHandler01_OuterDuplicatebErrorTrue');



fbCaseTest0601(
	bExecute:= TRUE, 
	bIsDuplicateOuters:= TRUE, 
	bIsDuplicatePacks:= FALSE, 
	stCTDateTime:= stCTDateTime_tests, 
	stOuterDataNotFound:= stRejectReasonsForOuter_tests.stOuterDataNotFound, 
	stProductInstruction:= stProductInstruction_test_0601, 
	nSecquentionalCounter:= nSecquentionalCounter_tests, 
	stCodeInfo_Outer:= stCodeInfo_Outer_tests, 
	stCaseRejectReasons:= stCaseRejectReasons_tests, 
	stCACData:= stCACData_test_0601, 
	bDone=> bDone, 
	bBusy=> bBusy, 
	bError=> bError, 
	nErrorID=> nErrorID, 
	sRejectCode=> sRejectCode_tets, 
	nValidationIndex=> nValidationIndex
);
	
rTrig(CLK:= fbCaseTest0601.bDone);
nCycles := nCycles + 1;	

IF rTrig.Q THEN	
		
	AssertEquals_BOOL(Expected 	:= TRUE,
					  Actual 	:= bError,
					  Message 	:= 'Outer duplicate did not call error'
	);
	
	AssertEquals_UDINT(Expected := 1,
                   	   Actual 	:= fbCaseTest0601.nErrorID,
                   	   Message 	:= 'Wrong nErrorID on outer duplicate'
	);
	
	TEST_FINISHED();
	
ELSIF nCycles > 50 THEN
	
	AssertTrue(Condition := TRUE,
			   Message 	 := 'Timeout duplicateHandler01_OuterDuplicatebErrorTrue'
	);	 
	TEST_FINISHED();
END_IF
END_METHOD

METHOD INTERNAL duplicateHandler02_PackDuplicatebErrorTrue
VAR
	//fbCaseTest			: FB_CASE_ValidateContent;
	bDone				: BOOL;
	bBusy				: BOOL;
	bError				: BOOL;
	nErrorID 			: UDINT;
	nValidationIndex	: INT;
	
	eLastState			: E_CAC_State;
			
END_VAR

VAR_INST
	fbCaseTest0602				: FB_CASE_ValidateContent;
	fTrig						: F_TRIG;	
	rTrig						: R_TRIG;
	nCycles						: INT;
	
END_VAR

//Data initialization
TestInit(stCACData:= stCACData_test_0602, stProductInstruction:= stProductInstruction_test_0602);

//Change some data for test scenario below

	
TcUnit.TEST('duplicateHandler02_PackDuplicatebErrorTrue');


fbCaseTest0602(
	bExecute:= TRUE, 
	bIsDuplicateOuters:= FALSE, 
	bIsDuplicatePacks:= TRUE, 
	stCTDateTime:= stCTDateTime_tests, 
	stOuterDataNotFound:= stRejectReasonsForOuter_tests.stOuterDataNotFound, 
	stProductInstruction:= stProductInstruction_test_0602, 
	nSecquentionalCounter:= nSecquentionalCounter_tests, 
	stCodeInfo_Outer:= stCodeInfo_Outer_tests, 
	stCaseRejectReasons:= stCaseRejectReasons_tests, 
	stCACData:= stCACData_test_0602, 
	bDone=> bDone, 
	bBusy=> bBusy, 
	bError=> bError, 
	nErrorID=> nErrorID, 
	sRejectCode=> sRejectCode_tets, 
	nValidationIndex=> nValidationIndex
);
	
rTrig(CLK:= fbCaseTest0602.bDone);
nCycles := nCycles + 1;	

IF rTrig.Q THEN	
		
	AssertEquals_BOOL(Expected 	:= TRUE,
					  Actual 	:= bError,
					  Message 	:= 'Pack duplicate did not call error'
	);
	
	AssertEquals_UDINT(Expected := 1,
                   	   Actual 	:= fbCaseTest0602.nErrorID,
                   	   Message 	:= 'Wrong nErrorID on pack duplicate'
	);
	
	TEST_FINISHED();
	
ELSIF nCycles > 50 THEN
	
	AssertTrue(Condition := TRUE,
			   Message 	 := 'Timeout duplicateHandler02_PackDuplicatebErrorTrue'
	);	 
	TEST_FINISHED();
END_IF
END_METHOD

METHOD INTERNAL main01_bExecuteFalseNoAction
VAR
	//fbCaseTest			: FB_CASE_ValidateContent;
	bDone				: BOOL;
	bBusy				: BOOL;
	bError				: BOOL;
	nErrorID 			: UDINT;
	nValidationIndex	: INT;
	
	eLastState			: E_CAC_State;
			
END_VAR

VAR_INST
	fbCaseTest0101				: FB_CASE_ValidateContent;
	fTrig						: F_TRIG;	
	rTrig						: R_TRIG;
	nCycles						: INT;
	
END_VAR

//Data initialization
TestInit(stCACData:= stCACData_test_0101, stProductInstruction:= stProductInstruction_test_0101);

//Change some data for test scenario below

	
TcUnit.TEST('main01_bExecuteFalseNoAction');


fbCaseTest0101(
	bExecute:= FALSE, 
	bIsDuplicateOuters:= FALSE, 
	bIsDuplicatePacks:= FALSE, 
	stCTDateTime:= stCTDateTime_tests, 
	stOuterDataNotFound:= stRejectReasonsForOuter_tests.stOuterDataNotFound, 
	stProductInstruction:= stProductInstruction_test_0101, 
	nSecquentionalCounter:= nSecquentionalCounter_tests, 
	stCodeInfo_Outer:= stCodeInfo_Outer_tests, 
	stCaseRejectReasons:= stCaseRejectReasons_tests, 
	stCACData:= stCACData_test_0101, 
	bDone=> bDone, 
	bBusy=> bBusy, 
	bError=> bError, 
	nErrorID=> nErrorID, 
	sRejectCode=> sRejectCode_tets, 
	nValidationIndex=> nValidationIndex
);
	
rTrig(CLK:= fbCaseTest0101.bDone);
nCycles := nCycles + 1;	

		
AssertEquals_BOOL(Expected 	:= FALSE,
				  Actual 	:= fbCaseTest0101.bError,
				  Message 	:= 'FB no executed wrong output'
);

AssertEquals_BOOL(Expected 	:= FALSE,
				  Actual 	:= fbCaseTest0101.bDone,
				  Message 	:= 'B no executed wrong output'
);

TEST_FINISHED();
END_METHOD

METHOD INTERNAL numberOfOuters01_ValueToLittlebErrorTrue
VAR
	//fbCaseTest			: FB_CASE_ValidateContent;
	bDone				: BOOL;
	bBusy				: BOOL;
	bError				: BOOL;
	nErrorID 			: UDINT;
	nValidationIndex	: INT;
	
	eLastState			: E_CAC_State;
			
END_VAR

VAR_INST
	fbCaseTest0301				: FB_CASE_ValidateContent;
	fTrig0301						: F_TRIG;
	nCycles0301						: INT;
	
END_VAR

//Data initialization
TestInit(stCACData:= stCACData_test_0301, stProductInstruction:= stProductInstruction_test_0301);

//Change some data for test scenario below
stCACData_test_0301.NumberOfOuters := 45;
	


TcUnit.TEST('numberOfOuters01_ValueToLittlebErrorTrue');

fbCaseTest0301(
	bExecute:= TRUE, 
	bIsDuplicateOuters:= FALSE, 
	bIsDuplicatePacks:= FALSE, 
	stCTDateTime:= stCTDateTime_tests, 
	stOuterDataNotFound:= stRejectReasonsForOuter_tests.stOuterDataNotFound, 
	stProductInstruction:= stProductInstruction_test_0301, 
	nSecquentionalCounter:= nSecquentionalCounter_tests, 
	stCodeInfo_Outer:= stCodeInfo_Outer_tests, 
	stCaseRejectReasons:= stCaseRejectReasons_tests, 
	stCACData:= stCACData_test_0301, 
	bDone=> bDone, 
	bBusy=> bBusy, 
	bError=> bError, 
	nErrorID=> nErrorID, 
	sRejectCode=> sRejectCode_test_0301, 
	nValidationIndex=> nValidationIndex
);

fTrig0301(CLK:= fbCaseTest0301.bBusy);
nCycles0301 := nCycles0301 + 1;	

IF fTrig0301.Q AND nCycles0301 <= 50 THEN	
	
	AssertEquals_BOOL(Expected := TRUE,
					  Actual := fbCaseTest0301.bError,
					  Message := 'Numbers of outer wrong value didnt call error'
	);
	
	AssertEquals_STRING(Expected := 'XXVAL045XX',
						Actual := TO_STRING(fbCaseTest0301.sRejectCode),
						Message := 'Wrong value of nErrorID'
	);
	
	AssertEquals_INT(Expected := 45,
					 Actual := stCACData_test_0301.NumberOfOuters,
					 Message := 'INT Values differ'
	);	
	
	TEST_FINISHED();
	
ELSIF nCycles0301 > 50 THEN
	
	AssertTrue(Condition := TRUE,
			   Message := 'Timeout CASE loop within FB_CASE_Validation'
	);	 

	
	TEST_FINISHED();
END_IF
END_METHOD

METHOD INTERNAL numberOfOuters02_ValueGraterErrorTrue
VAR
	
	bDone				: BOOL;
	bBusy				: BOOL;
	bError				: BOOL;
	nErrorID 			: UDINT;
	nValidationIndex	: INT;
	
	eLastState			: E_CAC_State;
	
		
END_VAR

VAR_INST
	
	fbCaseTest0302				: FB_CASE_ValidateContent;
	fTrig0302						: F_TRIG;
	nCycles0302						: INT;
	
END_VAR

//Data initialization
TestInit(stCACData:= stCACData_test_0302, stProductInstruction:= stProductInstruction_test_0302);

//Change some data for test scenario below
stCACData_test_0302.NumberOfOuters := 79;

	
TcUnit.TEST('numberOfOuters02_ValueGraterErrorTrue');


fbCaseTest0302(
	bExecute:= TRUE, 
	bIsDuplicateOuters:= FALSE, 
	bIsDuplicatePacks:= FALSE, 
	stCTDateTime:= stCTDateTime_tests, 
	stOuterDataNotFound:= stRejectReasonsForOuter_tests.stOuterDataNotFound, 
	stProductInstruction:= stProductInstruction_test_0302, 
	nSecquentionalCounter:= nSecquentionalCounter_tests, 
	stCodeInfo_Outer:= stCodeInfo_Outer_tests, 
	stCaseRejectReasons:= stCaseRejectReasons_tests, 
	stCACData:= stCACData_test_0302, 
	bDone=> bDone, 
	bBusy=> bBusy, 
	bError=> bError, 
	nErrorID=> nErrorID, 
	sRejectCode=> sRejectCode_test_0302, 
	nValidationIndex=> nValidationIndex
);
	
fTrig0302(CLK:= fbCaseTest0302.bBusy);
nCycles0302 := nCycles0302 + 1;	

IF fTrig0302.Q AND nCycles0302 <= 50 THEN	
		
	AssertEquals_BOOL(Expected := TRUE,
					  Actual := fbCaseTest0302.bError,
					  Message := 'Numbers of outer wrong value didnt call error'
	);
	
	AssertEquals_STRING(Expected := 'XXVAL079XX',
						Actual := TO_STRING(fbCaseTest0302.sRejectCode),
						Message := 'Wrong value of sRejectCode'
	);
	
	TEST_FINISHED();
	
ELSIF nCycles0302 > 50 THEN
	
	AssertTrue(Condition := TRUE,
			   Message 	 := 'Timeout numberOfOuters02_ValueGraterErrorTrue'
	);	 
	
	TEST_FINISHED();
END_IF
END_METHOD

METHOD INTERNAL numberOfOuters03_ValueToLittlebErrorTrueRejectCodeWright
VAR
	//fbCaseTest			: FB_CASE_ValidateContent;
	bDone				: BOOL;
	bBusy				: BOOL;
	bError				: BOOL;
	nErrorID 			: UDINT;
	nValidationIndex	: INT;
	
	eLastState			: E_CAC_State;
			
END_VAR

VAR_INST
	fbCaseTest0303				: FB_CASE_ValidateContent;
	fTrig						: F_TRIG;
	nCycles						: INT;
	
END_VAR

//Data initialization
TestInit(stCACData:= stCACData_test_0303, stProductInstruction:= stProductInstruction_test_0303);

//Change some data for test scenario below
stCACData_test_0303.NumberOfOuters := 51;

	
TcUnit.TEST('numberOfOuters03_ValueToLittlebErrorTrueRejectCodeWright');


fbCaseTest0303(
	bExecute:= TRUE, 
	bIsDuplicateOuters:= FALSE, 
	bIsDuplicatePacks:= FALSE, 
	stCTDateTime:= stCTDateTime_tests, 
	stOuterDataNotFound:= stRejectReasonsForOuter_tests.stOuterDataNotFound, 
	stProductInstruction:= stProductInstruction_test_0301, 
	nSecquentionalCounter:= nSecquentionalCounter_tests, 
	stCodeInfo_Outer:= stCodeInfo_Outer_tests, 
	stCaseRejectReasons:= stCaseRejectReasons_tests, 
	stCACData:= stCACData_test_0303, 
	bDone=> bDone, 
	bBusy=> bBusy, 
	bError=> bError, 
	nErrorID=> nErrorID, 
	sRejectCode=> sRejectCode_test_0303, 
	nValidationIndex=> nValidationIndex
);
	
fTrig(CLK:= fbCaseTest0303.bBusy);
nCycles := nCycles + 1;	

IF fTrig.Q THEN	
		
	AssertEquals_BOOL(Expected := TRUE,
					  Actual := fbCaseTest0303.bError,
					  Message := 'Numbers of outer wrong value didnt call error'
	);
	
	AssertEquals_STRING(Expected := 'XXVAL051XX',
						Actual := TO_STRING(fbCaseTest0303.sRejectCode),
						Message := 'Wrong value of sRejectCode'
	);
	
	TEST_FINISHED();
	
ELSIF nCycles > 50 THEN
	
	AssertTrue(Condition := TRUE,
			   Message 	 := 'Timeout numberOfOuters03_ValueToLittlebErrorTrueRejectCodeWright'
	);	 
	
	TEST_FINISHED();
END_IF
END_METHOD

METHOD INTERNAL oacMissing01nErrorID21
VAR
	//fbCaseTest			: FB_CASE_ValidateContent;
	bDone				: BOOL;
	bBusy				: BOOL;
	bError				: BOOL;
	nErrorID 			: UDINT;
	nValidationIndex	: INT;
	bCompare			: BOOL;
	
	eLastState			: E_CAC_State;
			
END_VAR

VAR_INST
	fbCaseTest0701				: FB_CASE_ValidateContent;
	fTrig0701					: F_TRIG;	
	rTrig0701					: R_TRIG;
	nCycles0701					: INT;
	
END_VAR

//Data initialization
TestInit(stCACData:= stCACData_test_0701, stProductInstruction:= stProductInstruction_test_0701);

//Change some data for test scenario below
stCACData_test_0701.Outer[5].OuterRejectID := 207;
stProductInstruction_test_0701.nCaseAcceptanceLevelOuters := 60;
stProductInstruction_test_0701.nOuterAcceptanceLevelPacks := 100;
stProductInstruction_test_0701.nCaseAcceptanceLevelPacks  := 100;
	
TcUnit.TEST('oacMissing01nErrorID21');


fbCaseTest0701(
	bExecute:= TRUE, 
	bIsDuplicateOuters:= FALSE, 
	bIsDuplicatePacks:= FALSE, 
	stCTDateTime:= stCTDateTime_tests, 
	stOuterDataNotFound:= stRejectReasonsForOuter_tests.stOuterDataNotFound, 
	stProductInstruction:= stProductInstruction_test_0701, 
	nSecquentionalCounter:= nSecquentionalCounter_tests, 
	stCodeInfo_Outer:= stCodeInfo_Outer_tests, 
	stCaseRejectReasons:= stCaseRejectReasons_tests, 
	stCACData:= stCACData_test_0701, 
	bDone=> bDone, 
	bBusy=> bBusy, 
	bError=> bError, 
	nErrorID=> nErrorID, 
	sRejectCode=> sRejectCode_tets, 
	nValidationIndex=> nValidationIndex
);
	
rTrig0701(CLK:= fbCaseTest0701.bDone);
nCycles0701 := nCycles0701 + 1;	



IF rTrig0701.Q THEN	
	
	bCompare := (stCACData_test_0701.CaseRejectID = stCaseRejectReasons_tests.stOACError.nRejectID);
	
	AssertEquals_BOOL(Expected 	:= TRUE,
					  Actual 	:= bError,
					  Message 	:= 'Pack duplicate did not call error'
	);
	
	AssertEquals_UDINT(Expected := 21,
                   	   Actual 	:= fbCaseTest0701.nErrorID,
                   	   Message 	:= 'Wrong nErrorID on OAC missing'
	);
	
	AssertEquals_BOOL(Expected 	:= TRUE,
					  Actual 	:= bCompare,
					  Message 	:= 'CaseRejectID wrong value'
	);	
	
	TEST_FINISHED();
	
ELSIF nCycles0701 > 50 THEN
	
	AssertTrue(Condition := FALSE,
			   Message 	 := 'Timeout oacMissing01nErrorID21'
	);	 
	TEST_FINISHED();
END_IF
END_METHOD

METHOD INTERNAL outerAggrDissable01_sRejectCodeOK
VAR
	//fbCaseTest			: FB_CASE_ValidateContent;
	bDone				: BOOL;
	bBusy				: BOOL;
	bError				: BOOL;
	nErrorID 			: UDINT;
	nValidationIndex	: INT;
	
	eLastState			: E_CAC_State;
			
END_VAR

VAR_INST
	fbCaseTest0401				: FB_CASE_ValidateContent;
	rTrig0401					: R_TRIG;
	nCycles0401					: INT;
	
END_VAR

//Data initialization
TestInit(stCACData:= stCACData_test_0401, stProductInstruction:= stProductInstruction_test_0401);

//Change some data for test scenario below
stCACData_test_0401.CodingAndTrackingMode := 6;
	
TcUnit.TEST('outerAggrDissable01_sRejectCodeOK');


fbCaseTest0401(
	bExecute:= TRUE, 
	bIsDuplicateOuters:= FALSE, 
	bIsDuplicatePacks:= FALSE, 
	stCTDateTime:= stCTDateTime_tests, 
	stOuterDataNotFound:= stOuterDataNotFound_tests, 
	stProductInstruction:= stProductInstruction_test_0401, 
	nSecquentionalCounter:= nSecquentionalCounter_tests, 
	stCodeInfo_Outer:= stCodeInfo_Outer_tests, 
	stCaseRejectReasons:= stCaseRejectReasons_tests, 
	stCACData:= stCACData_test_0401, 
	bDone=> bDone, 
	bBusy=> bBusy, 
	bError=> bError, 
	nErrorID=> nErrorID, 
	sRejectCode=> sRejectCode_test_0401, 
	nValidationIndex=> nValidationIndex
);
	
rTrig0401(CLK:= fbCaseTest0401.bDone);
nCycles0401 := nCycles0401 + 1;	

IF rTrig0401.Q THEN	
	
	AssertEquals_STRING(Expected := 'OK',
						Actual := TO_STRING(fbCaseTest0401.sRejectCode),
						Message := 'Wrong value of nErrorID'
	);
	
	
	TEST_FINISHED();
	
ELSIF nCycles0401 > 50 THEN
	
	AssertTrue(Condition := TRUE,
			   Message 	 := 'Timeout outerAggrDissable01_sRejectCodeOK'
	);	 
	TEST_FINISHED();
END_IF
END_METHOD

METHOD INTERNAL outerAggrEnable01_PacksPerOuterZero
VAR
	//fbCaseTest			: FB_CASE_ValidateContent;
	bDone				: BOOL;
	bBusy				: BOOL;
	bError				: BOOL;
	nErrorID 			: UDINT;
	nValidationIndex	: INT;
	
	eLastState			: E_CAC_State;
			
END_VAR

VAR_INST
	fbCaseTest0501				: FB_CASE_ValidateContent;
	rTrig0501					: R_TRIG;
	nCycles0501					: INT;
	
END_VAR

//Data initialization
TestInit(stCACData:= stCACData_test_0501, stProductInstruction:= stProductInstruction_test_0501);

//Change some data for test scenario below
stCACData_test_0501.CodingAndTrackingMode := 8;
stProductInstruction_test_0501.nPacksPerOuter := 0;
	
TcUnit.TEST('outerAggrEnable01_PacksPerOuterZero');


fbCaseTest0501(
	bExecute:= TRUE, 
	bIsDuplicateOuters:= FALSE, 
	bIsDuplicatePacks:= FALSE, 
	stCTDateTime:= stCTDateTime_tests, 
	stOuterDataNotFound:= stRejectReasonsForOuter_tests.stOuterDataNotFound, 
	stProductInstruction:= stProductInstruction_test_0501, 
	nSecquentionalCounter:= nSecquentionalCounter_tests, 
	stCodeInfo_Outer:= stCodeInfo_Outer_tests, 
	stCaseRejectReasons:= stCaseRejectReasons_tests, 
	stCACData:= stCACData_test_0501, 
	bDone=> bDone, 
	bBusy=> bBusy, 
	bError=> bError, 
	nErrorID=> nErrorID, 
	sRejectCode=> sRejectCode_test_0501, 
	nValidationIndex=> nValidationIndex
);
	
rTrig0501(CLK:= fbCaseTest0501.bDone);
nCycles0501 := nCycles0501 + 1;	

IF rTrig0501.Q THEN	
	
	AssertEquals_BOOL(Expected 	:= TRUE,
					  Actual 	:= bError,
					  Message 	:= 'Wrong number of outers not detected'
	);

	AssertEquals_UDINT(Expected := 10,
                   	   Actual 	:= fbCaseTest0501.nErrorID,
                   	   Message 	:= 'nErrorID value wrong'
	);
	
	
	TEST_FINISHED();
	
ELSIF nCycles0501 > 50 THEN
	
	AssertTrue(Condition := TRUE,
			   Message 	 := 'Timeout outerAggrEnable01_PacksPerOuterZero'
	);	 
	TEST_FINISHED();
END_IF
END_METHOD

METHOD INTERNAL outerAggrEnable02_PacksPerCaseZero
VAR
	//fbCaseTest			: FB_CASE_ValidateContent;
	bDone				: BOOL;
	bBusy				: BOOL;
	bError				: BOOL;
	nErrorID 			: UDINT;
	nValidationIndex	: INT;
	
	eLastState			: E_CAC_State;
			
END_VAR

VAR_INST
	fbCaseTest0502				: FB_CASE_ValidateContent;
	rTrig0502					: R_TRIG;
	nCycles0502					: INT;
	
END_VAR

//Data initialization
TestInit(stCACData:= stCACData_test_0502, stProductInstruction:= stProductInstruction_test_0502);

//Change some data for test scenario below
stCACData_test_0502.CodingAndTrackingMode := 8;
stProductInstruction_test_0502.nPacksPerCase := 0;
	
TcUnit.TEST('outerAggrEnable02_PacksPerCaseZero');


fbCaseTest0502(
	bExecute:= TRUE, 
	bIsDuplicateOuters:= FALSE, 
	bIsDuplicatePacks:= FALSE, 
	stCTDateTime:= stCTDateTime_tests, 
	stOuterDataNotFound:= stRejectReasonsForOuter_tests.stOuterDataNotFound, 
	stProductInstruction:= stProductInstruction_test_0502, 
	nSecquentionalCounter:= nSecquentionalCounter_tests, 
	stCodeInfo_Outer:= stCodeInfo_Outer_tests, 
	stCaseRejectReasons:= stCaseRejectReasons_tests, 
	stCACData:= stCACData_test_0502, 
	bDone=> bDone, 
	bBusy=> bBusy, 
	bError=> bError, 
	nErrorID=> nErrorID, 
	sRejectCode=> sRejectCode_test_0502, 
	nValidationIndex=> nValidationIndex
);
	
rTrig0502(CLK:= fbCaseTest0502.bDone);
nCycles0502 := nCycles0502 + 1;	

IF rTrig0502.Q THEN	
	
	AssertEquals_BOOL(Expected 	:= TRUE,
					  Actual 	:= bError,
					  Message 	:= 'Wrong number of outers not detected'
	);

	AssertEquals_UDINT(Expected := 10,
                   	   Actual 	:= fbCaseTest0502.nErrorID,
                   	   Message 	:= 'nErrorID value wrong'
	);
	
	
	TEST_FINISHED();
	
ELSIF nCycles0502 > 50 THEN
	
	AssertTrue(Condition := TRUE,
			   Message 	 := 'Timeout outerAggrEnable02_PacksPerCaseZero'
	);	 
	TEST_FINISHED();
END_IF
END_METHOD

METHOD PRIVATE TestInit : BOOL
VAR_IN_OUT
	stProductInstruction	: ST_PCM_Status;
	stCACData 				: ST_CAC_Data;
END_VAR

VAR	
	rTrigDataInit		: R_TRIG;
	bDataInit			: BOOL;
	iOuter				: INT;
	iPack				: INT;
	sPackNum			: STRING;
	sOuterNum			: STRING;
	sPackCode			: STRING;
END_VAR

VAR_OUTPUT
	bDone				: BOOL;
END_VAR

//MEMSET(ADR(stCACData), 16#00, SIZEOF(stCACData));	

stProductInstruction.nOutersPerCase 	:= 50;
stProductInstruction.nPacksPerOuter		:= 10;
stProductInstruction.nPacksPerCase		:= 500;
stProductInstruction.nOpMode			:= 11;
stProductInstruction.sRetailSKU			:= '1234567';
stProductInstruction.nAcceptanceLevel 	:= 10;

stCACData.NumberOfOuters			:= stProductInstruction.nOutersPerCase;
stCACData.CodingAndTrackingMode		:= stProductInstruction.nOpMode;
stCACData.RetailSKU					:= stProductInstruction.sRetailSKU;

FOR iOuter := 1 TO stProductInstruction.nOutersPerCase DO
	(* Outer number z zerami *)
	sOuterNum := F_StringAddPrefix(INT_TO_STRING(iOuter),2,'0');

	stCACData.Outer[iOuter].Barcode    				:= CONCAT('OUTER', sOuterNum);
	stCACData.Outer[iOuter].NumberOfPacks 			:= stProductInstruction.nPacksPerOuter;
	stCACData.Outer[iOuter].NumberOfLinkedPacks 	:= stProductInstruction.nPacksPerOuter;
	stCACData.Outer[iOuter].AcceptanceLevel 		:= stProductInstruction.nAcceptanceLevel;
	stCACData.Outer[iOuter].CodingAndTrackingMode	:= stProductInstruction.nOpMode;
	stCACData.Outer[iOuter].OuterRejectCode			:= 'OK';

	FOR iPack := 1 TO stProductInstruction.nPacksPerOuter DO
		(* Pack number dwucyfrowy z zerami *)
		sPackNum := F_StringAddPrefix(INT_TO_STRING(iPack),2,'0');			
		(* Sklej pack code *)
		sPackCode := CONCAT(CONCAT('PACK', sPackNum), CONCAT('OUTER', sOuterNum));
		
		(* Write Pack Barcodes / Data*)
		stCACData.Outer[iOuter].PackCode[iPack]				:= sPackCode;
		stCACData.Outer[iOuter].PackCodeStatus[iPack]		:= 5;
		stCACData.Outer[iOuter].PackRejectID[iPack]			:= 0;			
		stCACData.Outer[iOuter].PackRejectCode[iPack]		:= 'OK';			
		stCACData.Outer[iOuter].PackCodeStatus[iPack].5 	:= TRUE;
		
		
		IF iPack = 1 THEN
			stCACData.Outer[iOuter].AggregationCodes[1]	:= stCACData.Outer[iOuter].PackCode[iPack];
		END_IF
		IF iPack = 2 THEN
			stCACData.Outer[iOuter].AggregationCodes[2]	:= stCACData.Outer[iOuter].PackCode[iPack];
		END_IF
	END_FOR
END_FOR	

stCACData.Outer[3].OuterCodeStatus.5 	:= TRUE;
stCACData.Outer[4].OuterCodeStatus.5	:= TRUE;
END_METHOD

END_FUNCTION_BLOCK

// ---- POUs/FinaliseCaseData/FB_CASE_ValidateContent.TcPOU
FUNCTION_BLOCK FB_CASE_ValidateContent
VAR_INPUT
	bExecute 					: BOOL;
	stCTDateTime				: ST_SYSTEM_DateTime;	(* CaseTrace date/time structure *)
END_VAR
VAR_IN_OUT

	stProductInstruction		: ST_PCM_Status;
	nSecquentionalCounter		: UDINT;
	stCodeInfo_Outer			: ST_CodeInfo;
	stCaseRejectReasons			: ST_RejectReasonsForCase;
	stCACData 					: ST_CAC_Data;
END_VAR
VAR_OUTPUT
	bDone 						: BOOL;
	bBusy						: BOOL;
	bError						: BOOL;
	nErrorID 					: UDINT;

	sRejectCode					: T_MaxString;
	nValidationIndex			: INT;

END_VAR
VAR
	fbExecute						: R_TRIG;
	eState						: E_CAC_STATE;
	eErrorState					: E_CAC_STATE;

	(*nIndex						: INT;*)

	//bValQtyOver				: BOOL;

	(*fbValidateCaseLabel				: FB_CODE_ValidateExplicitCode;*)
	nOutGTIN					: INT;
	nOutBand					: INT;
	nRetailSKU					: INT;
	nSerialCode					: INT;
	nTotalInvalide				: INT;

	fbValidateOuter				: FB_CODE_ValidateExplicitCode;
	nValidOACData				: INT;

	(*fbValidatePack					: FB_CODE_ValidateExplicitCode;*)
	nOuterIndex					: INT;
	nPackIndex					: INT;
	nValidPackData					: INT;
	//nIndex2: T_PositiveINT;
	//nIndex3: T_PositiveINT;

	aStatusErrorVal					: ARRAY[0..10] OF STRING(10);
	aRejectCodePointer     		   	: ARRAY[0..10] OF STRING(10);
END_VAR

(* rising edge of bExecute *)
fbExecute(CLK:= bExecute);

CASE eState OF

	E_CAC_IDLE:

		(* validate stCACData *)
		IF fbExecute.Q THEN

			(* update outputs *)
			bDone := FALSE;
			bBusy := TRUE;
			bError := FALSE;
			nErrorID := 0;

			MEMSET(ADR(aStatusErrorVal), 16#00, SIZEOF(aStatusErrorVal));
			MEMSET(ADR(aRejectCodePointer), 16#00, SIZEOF(aRejectCodePointer));

			(* clear outputs *)
			sRejectCode 		:= '';
			nValidationIndex	:= 0;

			eState := E_CAC_VALIDATECASE;

		(* bExecute has been reset *)
		ELSIF bExecute = FALSE THEN

			(* clear outputs *)
			bDone := FALSE;
			bBusy := FALSE;
			bError := FALSE;

		END_IF

	(* validate Case data *)
	E_CAC_VALIDATECASE:

		(* Outers in Case is correct *)
		IF stCACData.NumberOfOuters = stProductInstruction.nOutersPerCase THEN

			(* Outer aggregation enabled *)
			IF stCACData.CodingAndTrackingMode >= 7 THEN

				eState := E_CAC_VALIDATEOUTER;

			(* OAC data disabled *)
			ELSE
				eState := E_CAC_DONE;
			END_IF

		(* invalid Case *)
		ELSE

			(* update status *)
			bError := TRUE;
			eErrorState := eState;

			(* no validation code read *)
			IF stCACData.NumberOfOuters = -1 THEN

				(* error code *)
				nErrorID := 11;

				(* reset nNumberOfOuters to 0 and generate reject string *)
				stCACData.NumberOfOuters := 0;

				stCACData.CaseRejectCode 	:= stCaseRejectReasons.stCaseNoCaseData.sMetsDisplayCode;
				stCACData.CaseRejectID 		:= stCaseRejectReasons.stCaseNoCaseData.nRejectID;
				
			(* validation code not found in sInfeedQueue *)
			ELSIF stCACData.NumberOfOuters = -2 THEN

				(* error code *)
				nErrorID := 12;

				(* reset nNumberOfOuters to 0 and generate reject string *)
				stCACData.NumberOfOuters := 0;

				aStatusErrorVal[0] 		:= F_StringAddPrefix(INT_TO_STRING(stCACData.NumberOfOuters),2,'0');
				aRejectCodePointer[0] 	:= 'nn';

				stCACData.CaseRejectCode 	:= F_CODE_AssignValToStringWithPrefix(stCaseRejectReasons.stValError.sMetsDisplayCode, aStatusErrorVal, aRejectCodePointer, 3, '0');
				stCACData.CaseRejectID 		:= stCaseRejectReasons.stValError.nRejectID;

				(*eState := E_CAC_DONE;*)

			ELSIF stCACData.NumberOfOuters = -3 THEN

				(* error code *)
				nErrorID := 13;

				(* reset nNumberOfOuters to 0 and generate reject string *)
				stCACData.NumberOfOuters := stProductInstruction.nOutersPerCase;

				aStatusErrorVal[0] 		:= F_StringAddPrefix(INT_TO_STRING(stCACData.NumberOfOuters),2,'0');
				aRejectCodePointer[0] 	:= 'nn';

				stCACData.CaseRejectCode 	:= F_CODE_AssignValToStringWithPrefix(stCaseRejectReasons.stValError.sMetsDisplayCode, aStatusErrorVal, aRejectCodePointer, 3, '0');
				stCACData.CaseRejectID 		:= stCaseRejectReasons.stValError.nRejectID;

				(*eState := E_CAC_DONE;*)

			(* incorrect number of Outers *)
			ELSE

				aStatusErrorVal[0] 		:= F_StringAddPrefix(INT_TO_STRING(stCACData.NumberOfOuters),2,'0');
				aRejectCodePointer[0] 	:= 'nn';

				stCACData.CaseRejectCode 	:= F_CODE_AssignValToStringWithPrefix(stCaseRejectReasons.stValError.sMetsDisplayCode, aStatusErrorVal, aRejectCodePointer, 3, '0');
				stCACData.CaseRejectID 		:= stCaseRejectReasons.stValError.nRejectID;

				(* >=1 Outer(s) missed by Infeed camera *)
				IF stCACData.NumberOfOuters < stProductInstruction.nOutersPerCase THEN

					(* error code *)
					nErrorID := 14;

				(* >=1 Outer(s) physically removed from Infeed queue *)
				ELSE
					(* error code *)
					nErrorID := 15;
				END_IF
			END_IF

			eState := E_CAC_DONE;
		END_IF

	(* validate RetailSKU for each Outer *)
	E_CAC_VALIDATEOUTER:

		(* initialise counters *)
		nOutGTIN		:= 0;
		nOutBand		:= 0;
		nRetailSKU 		:= 0;
		nSerialCode 	:= 0;
		nTotalInvalide	:= 0;

		(* for each Outer *)
		FOR nOuterIndex := 1 TO stCACData.NumberOfOuters DO

			fbValidateOuter(	sFullCode := stCACData.Outer[nOuterIndex].Barcode,
							stCodeInfo := stCodeInfo_Outer,
							stProductInstruction := stProductInstruction);

			IF fbValidateOuter.bGtinOK  THEN

				(* Outer has valid GTIN *)
				nOutGTIN := nOutGTIN + 1;
			END_IF

			IF fbValidateOuter.bBrandOK  THEN

				(* Outer has valid GTIN *)
				nOutBand := nOutBand + 1;
			END_IF

			IF fbValidateOuter.bSerialCodeOK  THEN

				(* Outer has valid SerialCode *)
				nSerialCode := nSerialCode + 1;
			END_IF

			IF fbValidateOuter.bRskuOK  THEN

				(* Outer has valid RetailSKU *)
				nRetailSKU := nRetailSKU + 1;
			END_IF

			IF fbValidateOuter.bValidationOK THEN

				(* Total number of invalide outers - whatever reaso*)
				nTotalInvalide := nTotalInvalide +1;
			END_IF
		END_FOR


		(* all Outers have valid GTIN *)
		IF  nOutGTIN = stProductInstruction.nOutersPerCase THEN
			(* all Outers have valid Brand *)
			IF  nOutBand = stProductInstruction.nOutersPerCase THEN
				(* all Outers have valid RetailSKU *)
				IF  nRetailSKU = stProductInstruction.nOutersPerCase  THEN
					(* all Outers have valid SerialCode *)
					IF  nSerialCode = stProductInstruction.nOutersPerCase THEN
						(*If total invalide Outers inside a case*)
						IF  nTotalInvalide = stProductInstruction.nOutersPerCase THEN
	
							eState := E_CAC_VALIDATEOAC;
	
						ELSE
							(* RejectCode *)
							bError := TRUE;
							nErrorID := 16;
							eErrorState := eState;

							aStatusErrorVal[0] 		:= F_StringAddPrefix(INT_TO_STRING(stCACData.NumberOfOuters - nTotalInvalide),2,'0');
							aRejectCodePointer[0] 	:= 'nn';
						
							stCACData.CaseRejectCode 	:= F_CODE_AssignValToStringWithPrefix(stCaseRejectReasons.stINVError.sMetsDisplayCode, aStatusErrorVal, aRejectCodePointer, 2, '0');
							stCACData.CaseRejectID 		:= stCaseRejectReasons.stINVError.nRejectID;
							
							eState := E_CAC_DONE;

						END_IF
					(* 1 or more Outers have incorrect SerialCode *)
					ELSE
		
						(* RejectCode *)
						bError := TRUE;
						nErrorID := 17;
						eErrorState := eState;
	
						(* generate reject string *)
	
						aStatusErrorVal[0] 		:= F_StringAddPrefix(INT_TO_STRING(stCACData.NumberOfOuters - nSerialCode),2,'0');
						aRejectCodePointer[0] 	:= 'nn';
	
						stCACData.CaseRejectCode 	:= F_CODE_AssignValToStringWithPrefix(stCaseRejectReasons.stOuterSerialError.sMetsDisplayCode, aStatusErrorVal, aRejectCodePointer, 2, '0');
						stCACData.CaseRejectID 		:= stCaseRejectReasons.stOuterSerialError.nRejectID;
					
						eState := E_CAC_DONE;
	
					END_IF
	
				(* 1 or more Outers with invalid RetailSKU *)
				ELSE
		
					(* RejectCode *)
					bError := TRUE;
					nErrorID := 18;
					eErrorState := eState;
		
					(* generate reject string *)
	
					aStatusErrorVal[0] 		:= F_StringAddPrefix(INT_TO_STRING(stCACData.NumberOfOuters - nRetailSKU),2,'0');
					aRejectCodePointer[0] 	:= 'nn';
		
					stCACData.CaseRejectCode 	:= F_CODE_AssignValToStringWithPrefix(stCaseRejectReasons.stOuterRSKUError.sMetsDisplayCode, aStatusErrorVal, aRejectCodePointer, 2, '0');
					stCACData.CaseRejectID 		:= stCaseRejectReasons.stOuterRSKUError.nRejectID;
					
					eState := E_CAC_DONE;
	
				END_IF
			ELSE
				(* RejectCode *)
				bError := TRUE;
				nErrorID := 19;
				eErrorState := eState;
	
				(* generate reject string *)

				aStatusErrorVal[0] 		:= F_StringAddPrefix(INT_TO_STRING(stCACData.NumberOfOuters - nOutBand),2,'0');
				aRejectCodePointer[0] 	:= 'nn';
	
				stCACData.CaseRejectCode 	:= F_CODE_AssignValToStringWithPrefix(stCaseRejectReasons.stOuterBrandError.sMetsDisplayCode, aStatusErrorVal, aRejectCodePointer, 2, '0');
				stCACData.CaseRejectID 		:= stCaseRejectReasons.stOuterBrandError.nRejectID;
				
				eState := E_CAC_DONE;
			END_IF
		ELSE
		(* RejectCode *)
			bError := TRUE;
			nErrorID := 20;
			eErrorState := eState;

			(* generate reject string *)

			aStatusErrorVal[0] 		:= F_StringAddPrefix(INT_TO_STRING(stCACData.NumberOfOuters - nOutGTIN),2,'0');
			aRejectCodePointer[0] 	:= 'nn';

			stCACData.CaseRejectCode 	:= F_CODE_AssignValToStringWithPrefix(stCaseRejectReasons.stOuterGTINError.sMetsDisplayCode, aStatusErrorVal, aRejectCodePointer, 2, '0');
			stCACData.CaseRejectID 		:= stCaseRejectReasons.stOuterGTINError.nRejectID;
			
			eState := E_CAC_DONE;

		END_IF

(* check OAC data was loaded *)
	E_CAC_VALIDATEOAC:

		(* initialise counter *)
		nValidOACData := 0;

		(* for each Outer *)
		FOR nOuterIndex := 1 TO stCACData.NumberOfOuters DO

			IF stCACData.CodingAndTrackingMode = 7 THEN
				(* OAC mode >= CAC mode, OAC data will contain all data required for CAC mode *)
				IF  stCACData.Outer[nOuterIndex].DataSource <>  'NO_R' AND stCACData.Outer[nOuterIndex].CodingAndTrackingMode = stCACData.CodingAndTrackingMode  THEN
					(* count Outers with valid OAC data *)
					nValidOACData := nValidOACData + 1;
				END_IF
			ELSIF stCACData.CodingAndTrackingMode = 11 THEN
			(* CAC mode -> OAC data will contain all data required for CAC mode *)
				IF stCACData.Outer[nOuterIndex].DataSource <>  'NO_R'  AND stCACData.Outer[nOuterIndex].OuterRejectCode = 'OK'  THEN
					(* count Outers with valid OAC data *)
					nValidOACData := nValidOACData + 1;
				END_IF
			END_IF
		END_FOR

		(* all Outers with valid OAC data *)
		IF (nValidOACData *100 ) / stProductInstruction.nOutersPerCase   >=  stProductInstruction.nCaseAcceptanceLevelOuters THEN


			FOR nOuterIndex := 1 TO stCACData.NumberOfOuters DO

				IF stCACData.CodingAndTrackingMode >= 7 THEN
					(* CAC mode -> OAC data will contain all data required for CAC mode *)
						IF stCACData.Outer[nOuterIndex].DataSource =  'NO_R'  THEN

							stCACData.Outer[nOuterIndex].ProductionDate := F_StringWildcard('#YYYYMMDD#', stCTDateTime.sSystemTime);
							stCACData.Outer[nOuterIndex].ProductionTime := F_StringWildcard('#hhmmss#', stCTDateTime.sSystemTime);
							stCACData.Outer[nOuterIndex].ProductionTimeOffset := F_SYSTEM_SystemTimeOffsetToHHMM(stCTDateTime.nSystemTimeOffset);
		
							stCACData.Outer[nOuterIndex].OuterTimeStamp :=F_SYSTEM_SystemTimeAsISO8601(stCTDateTime.sSystemTime, stCTDateTime.sUTCTimeZoneOffset );
							stCACData.Outer[nOuterIndex].RetailSKU := stProductInstruction.sRetailSKU;
							stCACData.Outer[nOuterIndex].OuterMachine.ProductionSite :=  stProductInstruction.sProductionSite;
							stCACData.Outer[nOuterIndex].OuterMachine.ProductionLine := stProductInstruction.sProductionLine;
							stCACData.Outer[nOuterIndex].BatchNumber := stProductInstruction.sBatchNumber;
							stCACData.Outer[nOuterIndex].CodingAndTrackingMode := stProductInstruction.nOpMode;

							stCACData.Outer[nOuterIndex].NumberOfPacks	:=   stProductInstruction.nPacksPerOuter;
							stCACData.Outer[nOuterIndex].AcceptanceLevel	:= 	stProductInstruction.nAcceptanceLevel;

							stCACData.Outer[nOuterIndex].OuterRejectCode := 'OK';
							stCACData.Outer[nOuterIndex].OuterRejectID := 0;
							stCACData.Outer[nOuterIndex].DataSource :=  '3DC';

						ELSIF stCACData.Outer[nOuterIndex].DataSource <>  'NO_R'  AND stCACData.Outer[nOuterIndex].OuterRejectCode <> 'OK' THEN

							stCACData.Outer[nOuterIndex].OuterRejectCode := 'OK';
							stCACData.Outer[nOuterIndex].OuterRejectID := 0;
							stCACData.Outer[nOuterIndex].DataSource :=  '3DCR';
						END_IF
				END_IF
			END_FOR

			eState := E_CAC_VALIDATEPACK;

		(* 1 or more Outers with missing OAC data *)
		ELSE

			(* update status *)
			bError := TRUE;
			nErrorID := 21;
			eErrorState := eState;

			(* generate reject string *)

			aStatusErrorVal[0] 		:= F_StringAddPrefix(INT_TO_STRING(stCACData.NumberOfOuters - nValidOACData),2,'0');
			aRejectCodePointer[0] 	:= 'nn';

			stCACData.CaseRejectCode 	:= F_CODE_AssignValToStringWithPrefix(stCaseRejectReasons.stOACError.sMetsDisplayCode, aStatusErrorVal, aRejectCodePointer, 3, '0');
			stCACData.CaseRejectID 		:= stCaseRejectReasons.stOACError.nRejectID;

			eState := E_CAC_DONE;
		END_IF

	(* check that PackCode data is included with OAC data *)
	E_CAC_VALIDATEPACK:

		(* initialise counter *)
		nValidPackData := 0;

		(* for each Outer *)
		FOR nOuterIndex := 1 TO stCACData.NumberOfOuters DO

			(* count Outers with PackCode data - assume- outer reject station working fine and only good outers in case, NumberOfLinkedPacks= good pack  *)
			nValidPackData := nValidPackData + stCACData.Outer[nOuterIndex].NumberOfLinkedPacks ;

			FOR nPackIndex := 1 TO stCACData.Outer[nOuterIndex].NumberOfPacks DO

				IF stCACData.Outer[nOuterIndex].PackCodeStatus[nPackIndex].1
					AND stCACData.Outer[nOuterIndex].PackCodeStatus[nPackIndex].2
					AND stCACData.Outer[nOuterIndex].PackCodeStatus[nPackIndex].3	THEN

					nValidPackData := -1;
					EXIT;
				END_IF
			END_FOR

			IF nValidPackData = -1 THEN
				EXIT;
			END_IF

		END_FOR

		(* Outers with PackCode data is correct *)
		IF (nValidPackData *100 ) /  stProductInstruction.nPacksPerCase  >=   stProductInstruction.nCaseAcceptanceLevelPacks   THEN

			FOR nOuterIndex := 1 TO stCACData.NumberOfOuters DO

				IF stCACData.Outer[nOuterIndex].NumberOfLinkedPacks = 0 THEN
					stCACData.Outer[nOuterIndex].PackTimeStamp := F_SYSTEM_SystemTimeAsISO8601(stCTDateTime.sSystemTime, stCTDateTime.sUTCTimeZoneOffset );
				END_IF

				FOR nPackIndex := 1 TO stCACData.Outer[nOuterIndex].NumberOfPacks DO
					(*Tolerance do not modify NumberOfLinkedPacks per outer*) (*later, repalce with PackCodeStatus.0*)
					IF  stCACData.Outer[nOuterIndex].PackCode[nPackIndex] = '' THEN

						stCACData.Outer[nOuterIndex].PackCode[nPackIndex] := F_CODE_BATSerializator(stCTDateTime, ePack, TRUE, stProductInstruction, nSecquentionalCounter);
						(* change reject reason to adjust for tolerance *)
						(*additional bit passing to CAC*)
						stCACData.Outer[nOuterIndex].PackCodeStatus[nPackIndex]:=
														F_FiltredSetBitState16(TRUE, 'LOW', 4, TRUE, stCACData.Outer[nOuterIndex].PackCodeStatus[nPackIndex]);

						stCACData.Outer[nOuterIndex].PackRejectCode[nPackIndex] := 'OK';
						stCACData.Outer[nOuterIndex].PackRejectID[nPackIndex]	:= 0;
					END_IF
				END_FOR

				stCACData.Outer[nOuterIndex].NumberOfLinkedPacks := stCACData.Outer[nOuterIndex].NumberOfPacks;

			END_FOR

			eState := E_CAC_DONE;

		ELSIF nValidPackData = -1 THEN

			(* RejectCode *)
			bError := TRUE;
			nErrorID := 23;
			eErrorState := eState;
	
			aStatusErrorVal[0] 		:= 'PK';
			aRejectCodePointer[0] 	:= 'nn';

			stCACData.CaseRejectCode 	:= F_CODE_AssignValToStringWithPrefix(stCaseRejectReasons.stINVError.sMetsDisplayCode, aStatusErrorVal, aRejectCodePointer, 2, '0');
			stCACData.CaseRejectID 		:= stCaseRejectReasons.stINVError.nRejectID;

			eState := E_CAC_DONE;


		(* 1 or more Outers has no PackCode data *)
		ELSE

			(* update status *)
			bError := TRUE;
			nErrorID := 24;
			eErrorState := eState;

			(* generate reject string *)			(* generate reject string *)
			(*stCACData.RejectCode := F_CONCAT3('XXXPACK', F_StringAddPrefix(INT_TO_STRING(stCACData.NumberOfOuters - nValidPackData), 2, '0'), 'XXX');*)

			aStatusErrorVal[0] 		:= F_StringAddPrefix(INT_TO_STRING(stProductInstruction.nPacksPerCase - nValidPackData),2,'0');
			aRejectCodePointer[0] 	:= 'nn';

			stCACData.CaseRejectCode := F_CODE_AssignValToStringWithPrefix(stCaseRejectReasons.stPackNotLinedError.sMetsDisplayCode, aStatusErrorVal, aRejectCodePointer, 3, '0');
			stCACData.CaseRejectID 	 := stCaseRejectReasons.stPackNotLinedError.nRejectID;

			eState := E_CAC_DONE;
		END_IF

	(* complete *)
	E_CAC_DONE:

		(* no error found *)
		IF bError = FALSE THEN

			stCACData.CaseRejectCode 	:= 'OK';
			stCACData.CaseRejectID		:= 0;
		END_IF

		(* update outputs *)
		bBusy := FALSE;
		bDone := TRUE;
		sRejectCode := stCACData.CaseRejectCode;
		nValidationIndex := stCACData.NumberOfOuters;
		
		eState := E_CAC_IDLE;

(* unknown state *)
ELSE

	eState := E_CAC_IDLE;

	(* clear outputs *)
	bDone := FALSE;
	bBusy := FALSE;
	bError := FALSE;

END_CASE

END_FUNCTION_BLOCK

// ---- POUs/_Utilites/METS/Common LIB/08_SOFTWARE LIB/AI Codes And Validation FBs/F_CODE_AssignValToStringWithPrefix.TcPOU
FUNCTION F_CODE_AssignValToStringWithPrefix : T_MaxString
VAR_INPUT
	asRejectReason		: T_MaxString;
	anValue				: ARRAY[0..10] OF STRING(10);
	asPointer          	  		: ARRAY[0..10] OF STRING(10);
	nPrefixSize			: UINT;
	nPrefixValue			: STRING(5);
END_VAR

VAR
	(*bPointerNotFound	           : BOOL;*)
	nCounter				: INT;
	nPointerPos			: INT;
	asAssignedRejectReason	: T_MaxString;
	sValToAssign			: STRING(20);
END_VAR

(* This Function assigns value to predefined Pointer in string.
     Function can assing up to 10 Values
     For ex. string Reject Reason := 'XXDUPn1-n2XX'
     	         nValue := [3, 4], sPointer := ['n1', 'n2']		
	         asRejectReason := 'XXDUP3-4XX'	*)

F_CODE_AssignValToStringWithPrefix := '';

asAssignedRejectReason := asRejectReason;

REPEAT
	nPointerPos := FIND(asAssignedRejectReason, asPointer[nCounter]);
	IF nPointerPos > 0 AND  asPointer[nCounter] <> '' THEN
		sValToAssign :=  F_StringAddPrefix(anValue[nCounter], nPrefixSize, nPrefixValue);
		 asAssignedRejectReason := REPLACE(asAssignedRejectReason, sValToAssign, LEN(asPointer[nCounter]), nPointerPos);
	END_IF;
	nCounter := nCounter + 1;
UNTIL
	nCounter >= 10
END_REPEAT

IF nCounter <> 0 THEN
	F_CODE_AssignValToStringWithPrefix := asAssignedRejectReason;
ELSE
	F_CODE_AssignValToStringWithPrefix := asRejectReason;
END_IF;

END_FUNCTION

// ---- POUs/_Utilites/METS/F_StringWildcard.TcPOU
(* replaces date and time wildcards in string *)
FUNCTION F_StringWildcard : T_MaxString
VAR_INPUT
	strInput		: T_MaxString;	(* string with wildcard markers *)
	sDateTime		: TIMESTRUCT;	(* date/time structure *)
END_VAR
VAR
	fbExtractData	: FB_ExtractString;
	strWildcard		: T_MaxString;
	strData			: STRING(4);
	nCharPos		: INT;
END_VAR
VAR CONSTANT
	arrMonthCode	: ARRAY[0..12] OF STRING(1) :=[ '', 'A', 'B', 'C', 'D', 'E', 'F', 'G', 'H', 'I', 'J', 'K', 'L'];
END_VAR
(*
-------------------------------------------------------------------------------------------------
Date		Version	Author	Comments
-------------------------------------------------------------------------------------------------
13/04/2015	3.00.01	PB		Check for 'MM' and 'M' now checked last, fixes problem where 'M' followed by 'DD' during April will generate corrupt string.
30/01/2015	3.00.00	PB		Initial release.

-------------------------------------------------------------------------------------------------

The following wildcard strings are supported:
YYYY - Year (4 chars)				hh	- hour
YY	 - Year (last 2 chars)			mm	- minute
Y	 - Year (last char only)		ss	- second
MM	 - Month (01-12 = Jan-Dec)		t	- tenth of second
M	 - Month (A-L = Jan-Dec)
DD	 - Date
*)

(* find and extract wildcard string, enclosed by '#' chars *)
fbExtractData(
	bExtractData	:= TRUE,
	nExtractChars	:= 0, 
	strPrefix		:= '#',
	strSuffix		:= '#',
	strString		:= strInput
);

(* wildcard string found *)
IF fbExtractData.bStringFound = TRUE THEN

	(* log wildcard string for modification *)
	strWildcard := fbExtractData.strData;

	(* check for wildcard 'YYYY' *)
	nCharPos := FIND(strWildcard, 'YYYY');
	IF nCharPos > 0 THEN

		(* generate year as 4 chars and replace YYYY *)
		strData := F_StringAddPrefix(WORD_TO_STRING(sDateTime.wYear), 4, '0');
		strWildcard := REPLACE(strWildcard, strData, 4, nCharPos);

	(* wildcard 'YYYY' not found *)
	ELSE

		(* check for wildcard 'YY' *)
		nCharPos := FIND(strWildcard, 'YY');
		IF nCharPos > 0 THEN

			(* generate year as 2 chars and replace YY *)
			strData := F_StringAddPrefix(RIGHT(WORD_TO_STRING(sDateTime.wYear), 2), 2, '0');
			strWildcard := REPLACE(strWildcard, strData, 2, nCharPos);

		(* wildcard 'YY' not found *)
		ELSE
	
			(* check for wildcard 'Y' *)
			nCharPos := FIND(strWildcard, 'Y');
			IF nCharPos > 0 THEN
	
				(* generate year as 1 char and replace Y *)
				strData := RIGHT(WORD_TO_STRING(sDateTime.wYear), 1);
				strWildcard := REPLACE(strWildcard, strData, 1, nCharPos);
			END_IF
		END_IF
	END_IF

	(* check for wildcard 'DD' *)
	nCharPos := FIND(strWildcard, 'DD');
	IF nCharPos > 0 THEN

		(* generate date as 2 chars and replace DD *)
		strData := F_StringAddPrefix(WORD_TO_STRING(sDateTime.wDay), 2, '0');
		strWildcard := REPLACE(strWildcard, strData, 2, nCharPos);
	END_IF

	(* check for wildcard 'hh' *)
	nCharPos := FIND(strWildcard, 'hh');
	IF nCharPos > 0 THEN

		(* generate hour as 2 chars and replace hh *)
		strData := F_StringAddPrefix(WORD_TO_STRING(sDateTime.wHour), 2, '0');
		strWildcard := REPLACE(strWildcard, strData, 2, nCharPos);
	END_IF

	(* check for wildcard 'mm' *)
	nCharPos := FIND(strWildcard, 'mm');
	IF nCharPos > 0 THEN

		(* generate minute as 2 chars and replace mm *)
		strData := F_StringAddPrefix(WORD_TO_STRING(sDateTime.wMinute), 2, '0');
		strWildcard := REPLACE(strWildcard, strData, 2, nCharPos);
	END_IF

	(* check for wildcard 'ss' *)
	nCharPos := FIND(strWildcard, 'ss');
	IF nCharPos > 0 THEN

		(* generate second as 2 chars and replace ss *)
		strData := F_StringAddPrefix(WORD_TO_STRING(sDateTime.wSecond), 2, '0');
		strWildcard := REPLACE(strWildcard, strData, 2, nCharPos);
	END_IF

	(* check for wildcard 't' *)
	nCharPos := FIND(strWildcard, 't');
	IF nCharPos > 0 THEN

		(* generate tenth of second as 1 char and replace t *)
		strData := WORD_TO_STRING(sDateTime.wMilliseconds / 100);
		strWildcard := REPLACE(strWildcard, strData, 1, nCharPos);
	END_IF

	(* check for wildcard 'MM' *)
	nCharPos := FIND(strWildcard, 'MM');
	IF nCharPos > 0 THEN

		(* generate month as 2 chars and replace MM *)
		strData := F_StringAddPrefix(WORD_TO_STRING(sDateTime.wMonth), 2, '0');
		strWildcard := REPLACE(strWildcard, strData, 2, nCharPos);

	(* wildcard 'YYYY' not found *)
	ELSE

		(* check for wildcard 'M' *)
		nCharPos := FIND(strWildcard, 'M');
		IF nCharPos > 0 THEN

			(* generate month as 1 char and replace M *)
			strData := arrMonthCode[sDateTime.wMonth];
			strWildcard := REPLACE(strWildcard, strData, 1, nCharPos);
		END_IF
	END_IF

	(* insert strWildcard back into strInput *)
	F_StringWildcard := INSERT(strInput, strWildcard, TO_INT(fbExtractData.nStartPos) - 1);

(* no wildcard string found *)
ELSE

	(* strInput direct to output without modification *)
	F_StringWildcard := strInput;
END_IF

END_FUNCTION

// ---- POUs/_Utilites/METS/F_SYSTEM_SystemTimeOffsetToHHMM.TcPOU
(* generate time difference between local time and UTC as "+HH:MM" *)
FUNCTION F_SYSTEM_SystemTimeOffsetToHHMM : STRING(6)
VAR_INPUT
	nSystemTimeOffset	: DINT;		(* UTC offset in ms *)
END_VAR
VAR
	nHours				: DINT;
	nMins				: DINT;
END_VAR
(*
-------------------------------------------------------------------------------------------------
Date		Version	Author	Comments
-------------------------------------------------------------------------------------------------
01/08/2014	2.00.00	PB		Initial release

-------------------------------------------------------------------------------------------------
*)

(* convert ms to hours *)
nHours := ABS(nSystemTimeOffset) / 3600000;

(* remove hours and convert remaining ms to mins *)
nMins := (ABS(nSystemTimeOffset) MOD 3600000) / 60000;

(* construct output string as "+HH:MM" or "-HH:MM" *)
F_SYSTEM_SystemTimeOffsetToHHMM := F_CONCAT4(SEL(nSystemTimeOffset < 0, '+', '-'), F_StringAddPrefix(DINT_TO_STRING(nHours), 2, '0'), ':', F_StringAddPrefix(DINT_TO_STRING(nMins), 2, '0'));

END_FUNCTION

// ---- POUs/_Utilites/METS/Concat Function/F_CONCAT4.TcPOU
(* concatenate 4 strings *)
FUNCTION F_CONCAT4 : T_MaxString
VAR_INPUT
	strString1		: T_MaxString;
	strString2		: T_MaxString;
	strString3		: T_MaxString;
	strString4		: T_MaxString;
END_VAR
VAR
END_VAR
(*
-------------------------------------------------------------------------------------------------
Date		Version	Author	Comments
-------------------------------------------------------------------------------------------------
30/01/2015	3.00.00	PB		No change

-------------------------------------------------------------------------------------------------
05/02/2010	1.00.00	PB		Initial release

-------------------------------------------------------------------------------------------------
*)

F_CONCAT4 := CONCAT(strString1, strString2);
F_CONCAT4 := CONCAT(F_CONCAT4, strString3);
F_CONCAT4 := CONCAT(F_CONCAT4, strString4);

END_FUNCTION

// ---- POUs/_Utilites/METS/F_SYSTEM_SystemTimeAsISO8601.TcPOU
(* generate format 2018-08-08T11:46:15.4869506+02:00*)
FUNCTION F_SYSTEM_SystemTimeAsISO8601 : T_ISO8601Time
VAR_INPUT
	sSystemTime			: TIMESTRUCT;
	strUTCTimeZone		: STRING(6);
END_VAR
VAR
	strYear				: STRING(4);
	strMonth				: STRING(2);
	strDay				: STRING(2);
	strMiliseconds			: STRING(3);

	strHour				: STRING(2);
	strMinute				: STRING(2);
	strSecond				: STRING(2);

	strDate				: STRING(10);
	strTime				: STRING(13);

END_VAR

(*Date*)
	strYear:=F_StringAddPrefix(WORD_TO_STRING(sSystemTime.wYear), 4, '0');
	strMonth:=F_StringAddPrefix(WORD_TO_STRING(sSystemTime.wMonth), 2, '0');
	strDay:=F_StringAddPrefix(WORD_TO_STRING(sSystemTime.wDay), 2, '0');

(*Time*)
	strHour:=F_StringAddPrefix(WORD_TO_STRING(sSystemTime.wHour), 2, '0');
	strMinute:=F_StringAddPrefix(WORD_TO_STRING(sSystemTime.wMinute), 2, '0');
	strSecond:=F_StringAddPrefix(WORD_TO_STRING(sSystemTime.wSecond), 2, '0');
	strMiliseconds:=F_StringAddPrefix(WORD_TO_STRING(sSystemTime.wMilliseconds), 3, '0');
(*Print*)


	strDate:=F_CONCAT5(strYear, '-', strMonth, '-', strDay);
	strTime:=F_CONCAT6('T', strHour, ':', strMinute, ':', strSecond);
	strTime:=F_CONCAT3( strTime,'.', strMiliseconds);

	IF strUTCTimeZone = '+00:00' THEN
		F_SYSTEM_SystemTimeAsISO8601:=F_CONCAT3(strDate, strTime, 'Z');
	ELSE
		F_SYSTEM_SystemTimeAsISO8601:=F_CONCAT3(strDate, strTime, strUTCTimeZone);
	END_IF

END_FUNCTION

// ---- POUs/_Utilites/METS/Concat Function/F_CONCAT5.TcPOU
(* concatenate 5 strings *)
FUNCTION F_CONCAT5 : T_MaxString
VAR_INPUT
	strString1		: T_MaxString;
	strString2		: T_MaxString;
	strString3		: T_MaxString;
	strString4		: T_MaxString;
	strString5		: T_MaxString;
END_VAR
VAR
END_VAR
(*
-------------------------------------------------------------------------------------------------
Date		Version	Author	Comments
-------------------------------------------------------------------------------------------------
30/01/2015	3.00.00	PB		No change

-------------------------------------------------------------------------------------------------
05/02/2010	1.00.00	PB		Initial release

-------------------------------------------------------------------------------------------------
*)

F_CONCAT5 := CONCAT(strString1, strString2);
F_CONCAT5 := CONCAT(F_CONCAT5, strString3);
F_CONCAT5 := CONCAT(F_CONCAT5, strString4);
F_CONCAT5 := CONCAT(F_CONCAT5, strString5);

END_FUNCTION

// ---- POUs/_Utilites/METS/Concat Function/F_CONCAT6.TcPOU
(* concatenate 6 strings *)
FUNCTION F_CONCAT6 : T_MaxString
VAR_INPUT
	strString1		: T_MaxString;
	strString2		: T_MaxString;
	strString3		: T_MaxString;
	strString4		: T_MaxString;
	strString5		: T_MaxString;
	strString6		: T_MaxString;
END_VAR
VAR
END_VAR
(*
-------------------------------------------------------------------------------------------------
Date		Version	Author	Comments
-------------------------------------------------------------------------------------------------
30/01/2015	3.00.00	PB		No change

-------------------------------------------------------------------------------------------------
05/02/2010	1.00.00	PB		Initial release

-------------------------------------------------------------------------------------------------
*)

F_CONCAT6 := CONCAT(strString1, strString2);
F_CONCAT6 := CONCAT(F_CONCAT6, strString3);
F_CONCAT6 := CONCAT(F_CONCAT6, strString4);
F_CONCAT6 := CONCAT(F_CONCAT6, strString5);
F_CONCAT6 := CONCAT(F_CONCAT6, strString6);

END_FUNCTION

// ---- POUs/_Utilites/METS/Concat Function/F_CONCAT3.TcPOU
(* concatenate 3 strings *)
FUNCTION F_CONCAT3 : T_MaxString
VAR_INPUT
	strString1		: T_MaxString;
	strString2		: T_MaxString;
	strString3		: T_MaxString;
END_VAR
VAR
END_VAR
(*
-------------------------------------------------------------------------------------------------
Date		Version	Author	Comments
-------------------------------------------------------------------------------------------------
30/01/2015	3.00.00	PB		No change

-------------------------------------------------------------------------------------------------
05/02/2010	1.00.00	PB		Initial release

-------------------------------------------------------------------------------------------------
*)

F_CONCAT3 := CONCAT(strString1, strString2);
F_CONCAT3 := CONCAT(F_CONCAT3, strString3);

END_FUNCTION

// ---- POUs/_Utilites/METS/F_FiltredSetBitState16.TcPOU
(* updates state of specified bit in nWord value *)
FUNCTION F_FiltredSetBitState16 : WORD
VAR_INPUT
	bEnable		: BOOL;		(* set TRUE to update state of target bit in nValue *)
	sFiltrType		: STRING(5);
	nTargetBit		: INT;		(* bit number of bit to be updated (0-15) *)
	nSetState		: BOOL;		(* state to which nTargetBit should be set *)
	nValue			: WORD;	(* value in which target bit should be updated *)
END_VAR
VAR
	nMaskValue	: WORD;
END_VAR

(* bit update is enabled *)
IF bEnable = TRUE THEN

	IF sFiltrType = 'LOW' THEN
		nValue :=  nValue AND 16#FF00;
	ELSIF sFiltrType = 'HIGH' THEN
		nValue :=  nValue AND 16#00FF;
	ELSIF sFiltrType = 'ALL' THEN
		nValue :=  nValue AND 16#0000;
	END_IF

	(* target bit must be 0-15 *)
	IF nTargetBit <= 15 THEN

		(* calculate mask value from specified target bit *)
		nMaskValue := LREAL_TO_WORD(EXPT(2, nTargetBit));

		nValue := (nValue AND NOT nMaskValue) + (BOOL_TO_WORD(nSetState) * nMaskValue);

	(* target bit out of range *)
	ELSE

		nValue := nValue;
	END_IF

(* bit update disabled *)
ELSE

	nValue :=  nValue AND 16#0000;
END_IF

F_FiltredSetBitState16 := nValue;

END_FUNCTION

// ---- POUs/TcUnit/FB_CASE_DuplicatCheckTests/PRG_CASE_DuplicatCheckManual.TcPOU
PROGRAM PRG_CASE_DuplicatCheckManual
VAR
	fbCase_DuplicatCheck		: FB_CASE_DuplicatCheck;
	
	(* Init function/method declarations*)
	rTrigDataInit		: R_TRIG;
	bDataInit			: BOOL;
	iOuter				: INT;
	iPack				: INT;
	sPackNum			: STRING;
	sOuterNum			: STRING;
	sPackCode			: STRING;
	
	(* Inputs *)
	bExecute							: BOOL;
	
	(* In/Out *)
	stProductInstruction				: ST_PCM_Status;
	stOuterBarcodeDuplicate				: ST_RejectItems;
	stOuterDuplicatedPackCodesFound		: ST_RejectItems;
	stCaseRejectReasons					: ST_RejectReasonsForCase;
	stRejectReasonForOuters				: ST_RejectReasonsForOuter;	
	stRejectReasonForPacks				: ST_RejectReasonsForPack;	
	
	stCACData 							: ST_CAC_Data;
	
	(* Outputs *)	
	bDone 					: BOOL;
	bBusy					: BOOL;

	bCACValid				: BOOL;
	sRejectCode				: T_MaxString;
	bIsDuplicateOuters		: BOOL;
	bIsDuplicatePacks		: BOOL;
	bReadyToValidate		: BOOL;
	
	stUpdateCACData 		: ST_CAC_Data;
	
	
END_VAR

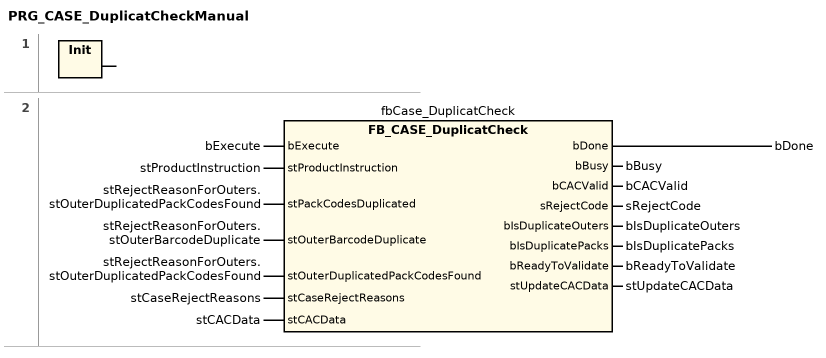
// NETWORK 1
Init();

// NETWORK 2
fbCase_DuplicatCheck(
    bExecute := bExecute,
    stProductInstruction := stProductInstruction,
    stPackCodesDuplicated := stRejectReasonForOuters.stOuterDuplicatedPackCodesFound,
    stOuterBarcodeDuplicate := stRejectReasonForOuters.stOuterBarcodeDuplicate,
    stOuterDuplicatedPackCodesFound := stRejectReasonForOuters.stOuterDuplicatedPackCodesFound,
    stCaseRejectReasons := stCaseRejectReasons,
    stCACData := stCACData,
    bBusy => bBusy,
    bCACValid => bCACValid,
    sRejectCode => sRejectCode,
    bIsDuplicateOuters => bIsDuplicateOuters,
    bIsDuplicatePacks => bIsDuplicatePacks,
    bReadyToValidate => bReadyToValidate,
    stUpdateCACData => stUpdateCACData); // FB_CASE_DuplicatCheck
bDone := fbCase_DuplicatCheck.bDone;

ACTION Init:

rTrigDataInit(CLK := bDataInit);

IF rTrigDataInit.Q THEN
	
stProductInstruction.nOutersPerCase		:= 50;
stProductInstruction.nPacksPerOuter 	:= 10;

	FOR iOuter := 1 TO stProductInstruction.nOutersPerCase DO
		(* Outer number z zerami *)
		sOuterNum := F_StringAddPrefix(INT_TO_STRING(iOuter),2,'0');
		
		(* Write Outers barcodes *)
		stCACData.Outer[iOuter].Barcode    := CONCAT('OUTER', sOuterNum);
		stCACData.Outer[iOuter].OuterCodeStatus := 5;
		
		FOR iPack := 1 TO stProductInstruction.nPacksPerOuter DO
			(* Pack number dwucyfrowy z zerami *)
			sPackNum := F_StringAddPrefix(INT_TO_STRING(iPack),2,'0');			
			(* Sklej pack code *)
			sPackCode := CONCAT(CONCAT('PACK', sPackNum), CONCAT('OUTER', sOuterNum));
			
			(* Write Pack Barcodes *)
			stCACData.Outer[iOuter].PackCode[iPack]			:= sPackCode;
			stCACData.Outer[iOuter].PackCodeStatus[iPack]	:= 5;
			stCACData.Outer[iOuter].PackRejectID[iPack]		:= 0;
			
		END_FOR;
	END_FOR;	
	
END_IF
END_ACTION

END_PROGRAM

// ---- POUs/FinaliseCaseData/FB_CASE_DuplicatCheck.TcPOU
FUNCTION_BLOCK FB_CASE_DuplicatCheck
VAR_INPUT
	bExecute	: BOOL;
END_VAR
VAR_IN_OUT

	stProductInstruction				: ST_PCM_Status;
	
	stPackCodesDuplicated				: ST_RejectItems;
	stOuterBarcodeDuplicate				: ST_RejectItems;
	stOuterDuplicatedPackCodesFound		: ST_RejectItems;
	stCaseRejectReasons					: ST_RejectReasonsForCase;
	
	stCACData 							: ST_CAC_Data;
END_VAR
VAR_OUTPUT
	bDone 					: BOOL;
	bBusy					: BOOL;

	bCACValid				: BOOL;
	sRejectCode				: T_MaxString;
	bIsDuplicateOuters		: BOOL;
	bIsDuplicatePacks		: BOOL;
	bReadyToValidate		: BOOL;
	
	stUpdateCACData 		: ST_CAC_Data;
END_VAR
VAR

	rtExecute	: R_TRIG;
	
	nOuterIndex			: INT;
	nPackIndex			: INT;
	nOuterCheckIndex	: INT;
	nPackCheckIndex		: INT;
	
	nDuplicateOuter1_Position	: INT;
	nDuplicateOuter2_Position	: INT;
	nDuplicatePack1_Position	: INT;
	nDuplicatePack2_Position	: INT;
	
	aStatusErrorVal					: ARRAY[0..10] OF STRING(10);
	aRejectCodePointer     		   	: ARRAY[0..10] OF STRING(10);
	
	nIteration				: UDINT;
	nIterationAI			: UDINT;
END_VAR

rtExecute(CLK:=bExecute);

IF rtExecute.Q THEN
	
	(* update outputs *)
	bDone := TRUE;
	bBusy := TRUE;

	bIsDuplicateOuters:= FALSE;
	bIsDuplicatePacks:= FALSE;
	
	MEMSET(ADR(aStatusErrorVal), 16#00, SIZEOF(aStatusErrorVal));
	MEMSET(ADR(aRejectCodePointer), 16#00, SIZEOF(aRejectCodePointer));
	
	bReadyToValidate	:= FALSE;
	MEMSET(ADR(stUpdateCACData), 16#00, SIZEOF(stUpdateCACData));
	

	nDuplicateOuter1_Position :=0;
	nDuplicateOuter2_Position:=0;
	nDuplicatePack1_Position:=0;
	nDuplicatePack2_Position:=0;

	(* clear outputs *)
	bCACValid := FALSE;
	sRejectCode := '';
	
	nIteration		:= 0;
	nIterationAI	:= 0;
(*
	(* Loop throught all packs in one case 'stCase' *)
	FOR nOuterIndex := 1 TO MIN(stProductInstruction.nOutersPerCase,cMAX_OUTERS_PER_CASE) BY 1 DO
		FOR nPackIndex := 1 TO MIN(stProductInstruction.nPacksPerOuter, cMAX_PACKS_PER_OUTER) BY 1 DO			
			(* Looking for same pack codes in all outers *)
			FOR nOuterCheckIndex := nOuterIndex TO MIN(stProductInstruction.nOutersPerCase,cMAX_OUTERS_PER_CASE) BY 1 DO
				
				IF stCACData.Outer[nOuterIndex].Barcode = stCACData.Outer[nOuterCheckIndex].Barcode AND 
					stCACData.Outer[nOuterIndex].Barcode <> ''										AND 
					NOT (nOuterCheckIndex = nOuterIndex) 											THEN
				 
					IF NOT bIsDuplicateOuters THEN
						nDuplicateOuter1_Position := nOuterIndex;
						nDuplicateOuter2_Position := nOuterCheckIndex;
					END_IF
						
					bIsDuplicateOuters := TRUE; 
					
					stCACData.Outer[nOuterIndex].OuterRejectCode 	:=	stOuterBarcodeDuplicate.sMetsDisplayCode;
					stCACData.Outer[nOuterIndex].OuterRejectID		:=	stOuterBarcodeDuplicate.nRejectID;
		
					stCACData.Outer[nOuterCheckIndex].OuterRejectCode 	:=	stOuterBarcodeDuplicate.sMetsDisplayCode;
					stCACData.Outer[nOuterCheckIndex].OuterRejectID		:=	stOuterBarcodeDuplicate.nRejectID;
				END_IF
				
				FOR nPackCheckIndex := 1 TO MIN(stProductInstruction.nPacksPerOuter, cMAX_PACKS_PER_OUTER) BY 1 DO
					nIterationAI := nIterationAI + 1;					
					(* Exclude comparing same pack with itself *)
					IF stCACData.Outer[nOuterIndex].PackCode[nPackIndex] = stCACData.Outer[nOuterCheckIndex].PackCode[nPackCheckIndex] 	AND 
						stCACData.Outer[nOuterIndex].PackCode[nPackIndex]  <> ''														AND 
						stCACData.Outer[nOuterCheckIndex].PackRejectID[nPackCheckIndex] <> stPackCodesDuplicated.nRejectID 				AND 
						NOT ((nOuterCheckIndex = nOuterIndex) AND (nPackCheckIndex = nPackIndex)) 										THEN
						
						IF NOT bIsDuplicatePacks AND NOT bIsDuplicateOuters THEN
							nDuplicateOuter1_Position := nOuterIndex;
							nDuplicateOuter2_Position :=  nOuterCheckIndex;
							nDuplicatePack1_Position := nPackIndex;
							nDuplicatePack2_Position := nPackCheckIndex;
						END_IF
							
						bIsDuplicatePacks := TRUE;
						stCACData.Outer[nOuterIndex].OuterRejectCode 	:= stOuterDuplicatedPackCodesFound.sMetsDisplayCode;
						stCACData.Outer[nOuterIndex].OuterRejectID		:= stOuterDuplicatedPackCodesFound.nRejectID;
						
						stCACData.Outer[nOuterCheckIndex].OuterRejectCode 	:= stOuterDuplicatedPackCodesFound.sMetsDisplayCode;
						stCACData.Outer[nOuterCheckIndex].OuterRejectID		:= stOuterDuplicatedPackCodesFound.nRejectID;
						
						stCACData.Outer[nOuterIndex].PackCodeStatus[nPackIndex] :=
											F_FiltredSetBitState16(TRUE, 'LOW', 3, TRUE, stCACData.Outer[nOuterIndex].PackCodeStatus[nPackIndex]);
						
						stCACData.Outer[nOuterIndex].PackRejectCode[nPackIndex]		:= stPackCodesDuplicated.sMetsDisplayCode;
						stCACData.Outer[nOuterIndex].PackRejectID[nPackIndex]		:= stPackCodesDuplicated.nRejectID;
						
						stCACData.Outer[nOuterCheckIndex].PackCodeStatus[nPackCheckIndex] :=
											F_FiltredSetBitState16(TRUE, 'LOW', 3, TRUE, stCACData.Outer[nOuterCheckIndex].PackCodeStatus[nPackCheckIndex]);
						
						stCACData.Outer[nOuterCheckIndex].PackRejectCode[nPackCheckIndex]	:= stPackCodesDuplicated.sMetsDisplayCode;
						stCACData.Outer[nOuterCheckIndex].PackRejectID[nPackCheckIndex]		:= stPackCodesDuplicated.nRejectID;
					END_IF
				END_FOR
			END_FOR			
		END_FOR
	END_FOR
	*)

//////////////////////	
	FOR nOuterIndex := 1 TO MIN(stProductInstruction.nOutersPerCase,cMAX_OUTERS_PER_CASE) BY 1 DO
	//////////////////////		
		FOR nOuterCheckIndex := nOuterIndex + 1 TO MIN(stProductInstruction.nOutersPerCase,cMAX_OUTERS_PER_CASE) BY 1 DO
			
			IF stCACData.Outer[nOuterIndex].Barcode = stCACData.Outer[nOuterCheckIndex].Barcode AND 
				stCACData.Outer[nOuterIndex].Barcode <> ''	THEN
	
			 	IF NOT bIsDuplicateOuters THEN
					nDuplicateOuter1_Position := nOuterIndex;
					nDuplicateOuter2_Position := nOuterCheckIndex;
				END_IF
					
				bIsDuplicateOuters := TRUE; 
				
				stCACData.Outer[nOuterIndex].OuterRejectCode 	:=	stOuterBarcodeDuplicate.sMetsDisplayCode;
				stCACData.Outer[nOuterIndex].OuterRejectID		:=	stOuterBarcodeDuplicate.nRejectID;
	
				stCACData.Outer[nOuterCheckIndex].OuterRejectCode 	:=	stOuterBarcodeDuplicate.sMetsDisplayCode;
				stCACData.Outer[nOuterCheckIndex].OuterRejectID		:=	stOuterBarcodeDuplicate.nRejectID;
			 END_IF
			 nIteration := nIteration + 1;
		END_FOR
		///////////////////////////
		FOR  nPackIndex :=1 TO MIN(stProductInstruction.nPacksPerOuter, cMAX_PACKS_PER_OUTER) BY 1 DO
			FOR nPackCheckIndex := nPackIndex + 1  TO MIN(stProductInstruction.nPacksPerOuter, cMAX_PACKS_PER_OUTER) BY 1 DO
				
				IF stCACData.Outer[nOuterIndex].PackCode[nPackIndex] = stCACData.Outer[nOuterIndex].PackCode[nPackCheckIndex] AND 
					stCACData.Outer[nOuterIndex].PackCode[nPackIndex]  <> ''										AND 
					stCACData.Outer[nOuterIndex].PackRejectID[nPackCheckIndex] <> stPackCodesDuplicated.nRejectID 	THEN
					
					IF NOT bIsDuplicatePacks AND NOT bIsDuplicateOuters THEN
						nDuplicateOuter1_Position := nOuterIndex;
						nDuplicateOuter2_Position :=  nOuterIndex;
						nDuplicatePack1_Position := nPackIndex;
						nDuplicatePack2_Position := nPackCheckIndex;
					END_IF
						
					bIsDuplicatePacks := TRUE;
					stCACData.Outer[nOuterIndex].OuterRejectCode 	:= stOuterDuplicatedPackCodesFound.sMetsDisplayCode;
					stCACData.Outer[nOuterIndex].OuterRejectID		:= stOuterDuplicatedPackCodesFound.nRejectID;
					
					stCACData.Outer[nOuterIndex].PackCodeStatus[nPackIndex] :=
											F_FiltredSetBitState16(TRUE, 'LOW', 3, TRUE, stCACData.Outer[nOuterIndex].PackCodeStatus[nPackIndex]);
											
					stCACData.Outer[nOuterIndex].PackRejectCode[nPackIndex]		:= stPackCodesDuplicated.sMetsDisplayCode;
					stCACData.Outer[nOuterIndex].PackRejectID[nPackIndex]		:= stPackCodesDuplicated.nRejectID;
					
					stCACData.Outer[nOuterIndex].PackCodeStatus[nPackCheckIndex] :=
											F_FiltredSetBitState16(TRUE, 'LOW', 3, TRUE, stCACData.Outer[nOuterIndex].PackCodeStatus[nPackCheckIndex]);
					
					stCACData.Outer[nOuterIndex].PackRejectCode[nPackCheckIndex]	:= stPackCodesDuplicated.sMetsDisplayCode;
					stCACData.Outer[nOuterIndex].PackRejectID[nPackCheckIndex]		:= stPackCodesDuplicated.nRejectID;
				END_IF
				nIteration := nIteration + 1;
			END_FOR
			/////////////////////////////////
			FOR nOuterCheckIndex := nOuterIndex + 1 TO MIN(stProductInstruction.nOutersPerCase,cMAX_OUTERS_PER_CASE) BY 1 DO
				FOR nPackCheckIndex := 1  TO MIN(stProductInstruction.nPacksPerOuter, cMAX_PACKS_PER_OUTER) BY 1 DO

					IF stCACData.Outer[nOuterIndex].PackCode[nPackIndex] = stCACData.Outer[nOuterCheckIndex].PackCode[nPackCheckIndex] AND 
						stCACData.Outer[nOuterIndex].PackCode[nPackIndex]  <> ''									AND 
						stCACData.Outer[nOuterCheckIndex].PackRejectID[nPackCheckIndex] <> stPackCodesDuplicated.nRejectID 	THEN
						
						IF NOT bIsDuplicatePacks AND NOT bIsDuplicateOuters THEN
							nDuplicateOuter1_Position := nOuterIndex;
							nDuplicateOuter2_Position :=  nOuterCheckIndex;
							nDuplicatePack1_Position := nPackIndex;
							nDuplicatePack2_Position := nPackCheckIndex;
						END_IF
							
						bIsDuplicatePacks := TRUE;
						stCACData.Outer[nOuterIndex].OuterRejectCode 	:= stOuterDuplicatedPackCodesFound.sMetsDisplayCode;
						stCACData.Outer[nOuterIndex].OuterRejectID		:= stOuterDuplicatedPackCodesFound.nRejectID;
						
						stCACData.Outer[nOuterCheckIndex].OuterRejectCode 	:= stOuterDuplicatedPackCodesFound.sMetsDisplayCode;
						stCACData.Outer[nOuterCheckIndex].OuterRejectID		:= stOuterDuplicatedPackCodesFound.nRejectID;
						
						stCACData.Outer[nOuterIndex].PackCodeStatus[nPackIndex] :=
											F_FiltredSetBitState16(TRUE, 'LOW', 3, TRUE, stCACData.Outer[nOuterIndex].PackCodeStatus[nPackIndex]);
						
						stCACData.Outer[nOuterIndex].PackRejectCode[nPackIndex]		:= stPackCodesDuplicated.sMetsDisplayCode;
						stCACData.Outer[nOuterIndex].PackRejectID[nPackIndex]		:= stPackCodesDuplicated.nRejectID;
						
						stCACData.Outer[nOuterCheckIndex].PackCodeStatus[nPackCheckIndex] :=
											F_FiltredSetBitState16(TRUE, 'LOW', 3, TRUE, stCACData.Outer[nOuterCheckIndex].PackCodeStatus[nPackCheckIndex]);
						
						stCACData.Outer[nOuterCheckIndex].PackRejectCode[nPackCheckIndex]	:= stPackCodesDuplicated.sMetsDisplayCode;
						stCACData.Outer[nOuterCheckIndex].PackRejectID[nPackCheckIndex]		:= stPackCodesDuplicated.nRejectID;
					END_IF
					nIteration := nIteration + 1;
				END_FOR
			END_FOR
		/////////////////////////////////		
		END_FOR
	//////////////////////	
	END_FOR
//////////////////////	


	IF bIsDuplicateOuters THEN
		
		aStatusErrorVal[0] := 	F_StringAddPrefix(INT_TO_STRING(nDuplicateOuter1_Position),2,'0');
		aStatusErrorVal[1] := 	F_StringAddPrefix(INT_TO_STRING(nDuplicateOuter2_Position),2,'0');
		aRejectCodePointer[0] := 'n1';
		aRejectCodePointer[1] := 'n2';
		
		stCACData.CaseRejectCode 	:=	F_CODE_AssignValToStringWithPrefix(stCaseRejectReasons.stDUPError.sMetsDisplayCode, aStatusErrorVal, aRejectCodePointer, 2, '0');
		stCACData.CaseRejectID	:= 	stCaseRejectReasons.stDUPError.nRejectID;
	
		sRejectCode := stCACData.CaseRejectCode;
		
	ELSIF bIsDuplicatePacks THEN
		
		aStatusErrorVal[0] := 	F_CONCAT4(F_StringAddPrefix(INT_TO_STRING(nDuplicateOuter1_Position),2,'0'),'(', F_StringAddPrefix(INT_TO_STRING(nDuplicatePack1_Position),2,'0'),')');
		aStatusErrorVal[1] := 	F_CONCAT4(F_StringAddPrefix(INT_TO_STRING(nDuplicateOuter2_Position),2,'0'),'(', F_StringAddPrefix(INT_TO_STRING(nDuplicatePack2_Position),2,'0'),')');
		aRejectCodePointer[0] := 'n1';
		aRejectCodePointer[1] := 'n2';

		stCACData.CaseRejectCode 	:=	F_CODE_AssignValToStringWithPrefix(stCaseRejectReasons.stDUPError.sMetsDisplayCode, aStatusErrorVal, aRejectCodePointer, 6, '0');
		stCACData.CaseRejectID		:= stCaseRejectReasons.stDUPError.nRejectID;
		
		sRejectCode := stCACData.CaseRejectCode;
	ELSE
		bCACValid := TRUE;
	END_IF
	
	bReadyToValidate	:= TRUE;
	MEMMOVE(ADR(stUpdateCACData), ADR(stCACData), SIZEOF(stUpdateCACData));
	
ELSIF bExecute = FALSE THEN
	
	(* clear outputs *)
	bDone := FALSE;
	bBusy := FALSE;

END_IF

END_FUNCTION_BLOCK

// ---- POUs/TcUnit/FB_CASE_DuplicateUpdateToDBTests/PRG_CASE_DuplicateUpdateToDBManual.TcPOU
PROGRAM PRG_CASE_DuplicateUpdateToDBManual
VAR
	fbCase_DuplicateUpdateToDB		: FB_CASE_DuplicateUpdateToDB;
	
	(* Data/Iterators for Init function/method *)
	rTrigDataInit			: R_TRIG;
	bDataInit				: BOOL;
	iOuter					: INT;
	iPack					: INT;
	sPackNum				: STRING;
	sOuterNum				: STRING;
	sPackCode				: STRING;
	stProductInstruction	: ST_PCM_Status;
	
	
	(* Inputs *)	
	bExecute						: BOOL;		(* set TRUE to archive OAC files *)
	bUseInterimCodeForValidation	: BOOL;
	
	
	(* In/Out *)
	aOCVPackStatus			: ARRAY[1..cMAX_OUTER_STATUS_QUEUE] OF ST_OUTER_Status;	(* Outer status array *)
	aOuterStatus			: ARRAY[1..cMAX_OUTER_STATUS_QUEUE] OF ST_OUTER_Status;	(* Outer status array *)
	
	stOCVDataDB							: ST_DB_OCVDataCtrl;
	stOACDataDB							: ST_DB_OACDataCtrl;
	
	stOuterBarcodeDuplicate				: ST_RejectItems;
	stOuterDuplicatedPackCodesFound		: ST_RejectItems;
	
	stCodeInfo_Pack				: ST_CodeInfo;
	stCodeInfo_Intermediate		: ST_CodeInfo;
	stCodeInfo_Outer			: ST_CodeInfo;
	
	stCACData					: ST_CAC_Data;
	
	(* Outputs *)
	bDone 					: BOOL;		(* TRUE = OAC archive complete *)
	bBusy 					: BOOL;		(* TRUE = OAC archive active *)
	bError 					: BOOL;		(* TRUE = OAC archive error *)
	nErrorID				: UDINT;	(* error code *)

	nOACFilesBlocked		: UINT;
	nOCVFilesBlocked		: UINT;
	stDaigOACDataDB			: ST_DB_OACDataCtrl;
	stDiagOCVDataDB			: ST_DB_OCVDataCtrl;
	
	
END_VAR

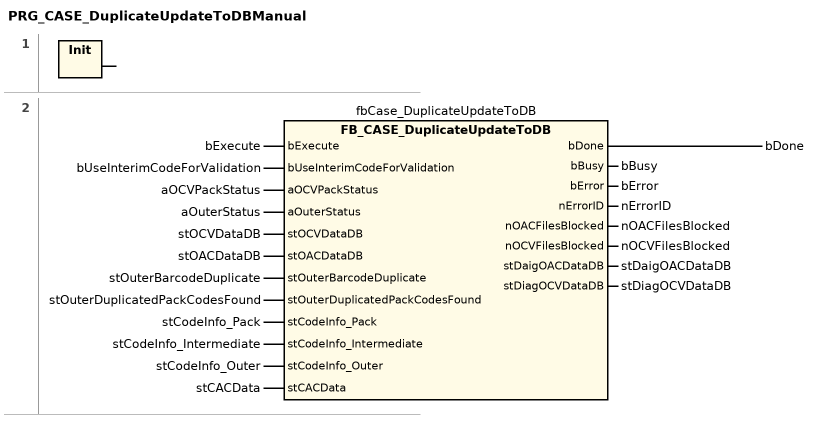
// NETWORK 1
Init();

